(* CODESYS project pmps3.5.0.library
   Company: SLAC - LCLS
   DefaultNamespace: PMPS
   Version: 3.5.0
   Description: Collection of PMPS functionality for LCLS PLCs
   Placeholder: PMPS
   Author: Alex Wallace and contributors
   Title: PMPS

Project tree, tasks and I/O mapping:
  libraries: LCLS General, * (SLAC); Tc2_MC2, * (Beckhoff Automation GmbH); Tc2_Standard, * (Beckhoff Automation GmbH); Tc2_System, * (Beckhoff Automation GmbH); Tc2_Utilities, * (Beckhoff Automation GmbH); Tc3_JsonXml, * (Beckhoff Automation GmbH); Tc3_Module, * (Beckhoff Automation GmbH); TcUnit, 1.2.0.0 (www.tcunit.org)
  AncillaryComponents/
    function block FB_JsonDocToSafeBP [ST]: ACT_FFO, ACT_Logger, M_LoadSafeBP
    function block FB_JsonFileToJsonDoc [ST]: ACT_FFO, ACT_Logger
    function block FB_PressSensor_FFO [ST]: ACT_Logger
    function block FB_TempSensor_FFO [ST]: ACT_Logger
  DUTs/
    InternalDUT/
      data type E_MPSBeamClasses
      data type E_MPSBeamRates
      data type K_Apertures
      data type K_Attenuators
      data type K_Stopper
      data type L_Apertures
      data type L_Attenuators
      data type L_Stopper
      data type ST_AttenuatorStatus
      data type ST_BP_ArbInternal
      data type ST_FF
      data type ST_FFInfo
      data type ST_FFOverride
      data type ST_PMPS_Aperture
      data type ST_PMPS_Attenuator
      data type T_HashTableEntry
    UserDUT/
      data type ST_BeamParams
      data type ST_DbStateParams
      data type ST_Device
      data type ST_ReactiveParams
    data type PMPS_CODES
    data type ST_DeviceState
    data type ST_DeviceStateExt
    data type ST_DeviceStateTable
  GVLs/
    global variables PMPS_GVL
    global variables PMPS_PARAM
    global variables PMPS_TOOLS
  HelperFunctions/
    TypeTranslators/
      function APT_TO_IO [ST]
      function ATT_TO_IO [ST]
      function BP_TO_IO [ST]
      function F_DeviceState_To_DeviceStateExt [ST]
      function IO_TO_APT [ST]
      function IO_TO_ATT [ST]
      function IO_TO_BP [ST]
    function F_AttenuatorOK [ST]
    function F_BPWithID [ST]
    function F_DifferentBeamParams [ST]
    function F_eVExcludeRange [ST]
    function F_eVIncludeRange [ST]
    function F_eVRangeCalculator [ST]
    function F_eVWithinSpec [ST]
    function F_InitTestBP [ST]
    function F_PMPS_JSON [ST]
    function F_SafeBPCompare [ST]
    function F_SafeBPCompare0Rate [ST]
    function F_SetBeamParams [ST]
    function F_SetGoodAttStatus [ST]
    function F_SetStateParams [ST]
    function F_ValidReqID [ST]
    function block FB_DummyArbIO [ST]: ApplyBPReq, AutoUpdateBP, CheckRequest, RemoveRequest, RequestBP, ElevateRequest, nLowerAuthorityID
    function block FB_DummyHA [ST]: CheckRequest, ElevateRequest, nLowerAuthorityID, RemoveRequest, RequestBP
    function block PE_Ranges [ST]: FB_init
  ImplicitChecks/
    function CheckBounds [ST]
    function CheckDivDInt [ST]
    function CheckDivLInt [ST]
    function CheckDivLReal [ST]
    function CheckDivReal [ST]
    function CheckLRangeSigned [ST]
    function CheckLRangeUnsigned [ST]
    function CheckPointer [ST]
    function CheckRangeSigned [ST]
    function CheckRangeUnsigned [ST]
  MajorComponents/
    Arbiter/
      function block FB_Arbiter [ST]: AddRequest, ArbitrateBP, CheckRequest, CheckRequestInPool, ElevateRequest, FB_init, GetArbitratedBP, nEntryCount, nLowerAuthorityID, RemoveRequest, RequestBP
      function block FB_BeamParamAssertionPool [ST]: A_Add, A_Count, A_GetFirst, A_GetNext, A_Lookup, A_Remove, A_Reset, DataPoolToEpics
      function block FB_VetoArbiter [ST]: CheckRequest, RemoveRequest, RequestBP
    BPTM/
      function block BeamParameterTransitionManager [ST]: AssertFinalBP, AssertTransitionBP, AuthorizeTransition, DeauthorizeTransition, LogActions, NewTarget_ENTRY, RemoveTransitionAssertion, RequestBP_DO, SetNewTarget, WaitingForFinalAssertion_DO, WaitingForFinalAssertion_EXIT, WaitingForTransitionAssertion_DO, WaitingForTransitionAssertion_EXIT
      data type E_BPTMState
    FastFaults/
      function block FB_FastFault [ST]
      function block FB_HardwareFFOutput [ST]: EvaluateOutput, EvaluateOverrides, EvaluateVetos, Execute, ExecuteLogging, ExecuteNoLog, FormulateLogJson, IdxCheckIn, Register
    InterPlcComm/
      function block FB_ArbiterToSubSys_IO [ST]
      function block FB_SubSysToArbiter_IO [ST]: CheckRequest, RemoveRequest, RequestBP
    PhotonEnergyInterface/
      function F_CalculatePhotonEnergy [ST]
      function block FB_AcceleratorLinks [ST]
      function block FB_Hgvpu [ST]: Init, rCurrentPhotonEnergy, rTargetPhotonEnergy, UndAdrUpdate
      function block FB_KPhotonEnergy [ST]
      function block FB_LPhotonEnergy [ST]
      function block FB_PhotonEnergy [ST]
      function block FB_SXU [ST]: Init, rCurrentPhotonEnergy, rTargetPhotonEnergy, UndAdrUpdate
      function block FB_UndulatorSegment [ST]
    PMPS_MPS_Interface/
      function block FB_BeamClassOutputs [ST]
      function block FB_BeamClassOutputs_BCD [ST]
      function block FB_BeamClassWatcher [ST]
      function block FB_CTLS_Outputs [ST]
      function block FB_MachineModeFromEPICS [ST]
      function block FB_PhotonEnergyWatcher [ST]
    SimulationFB/
      function block FB_eVSimulator [ST]
      function block FB_MachineSimulator [ST]
    Stoppers/
      function block FB_KStopper [ST]: FB_init
      function block FB_KVetoDevice [ST]: FB_init
      function block FB_LStopper [ST]: FB_init
      function block FB_LVetoDevice [ST]: FB_init
      function block FB_StopperWatcher [ST]
      function block FB_VetoDevice [ST]
    function block FB_BeamClassFromEPICS [ST]
    function block FB_BPControlDevice [ST]: FB_init
    function block FB_BPRequestor [ST]: CheckRequest, RemoveRequest, RequestBP
    function block FB_LinearDeviceStateTable [ST]: A_Add, A_Count, A_GetFirst, A_GetNext, A_Lookup, A_Remove, A_Reset
    function block FB_LinearGovernor [ST]
    function block FB_RateFromEPICS [ST]
    interface I_HigherAuthority: CheckRequest, RemoveRequest, RequestBP
    interface I_LowerAuthority: ElevateRequest, nLowerAuthorityID
    interface I_UndulatorComplex: rCurrentPhotonEnergy, rTargetPhotonEnergy
  TestComponents/
    DUT/
      data type E_ArbDosTestStates
      data type E_BPTMTestStates
    function block FB_Arbiter_Test [ST]: ArbiterCapacity, Arbitration, DoS, FullArbitrationStack, RemoveReq, RequestCheckRemoveBP, StackArbiters
    function block FB_ArbToSubsys_Test [ST]: BasicFunction
    function block FB_AttenuatorSimulator [ST]
    function block FB_BPTM_Test [ST]: BPTMBasicFunction, FullArbError, InterruptAtAllSteps
    function block FB_DiffBP_Test [ST]: BPDiff
    function block FB_evRangeCalculator_Test [ST]: BasicFunction
    function block FB_eVWithinSpec_Test [ST]: evWithinRangeChecks
    function block FB_FastFault_Test [ST]: FFCombinedFunctionality, FFOvrdAndNextFault, FFRegistration
    function block FB_PhotonEnergyWatcher_Test [ST]: PEWatcherBasicFunction
    function block FB_SafeBPCompare_Test [ST]: BeamOffIsSafe, BPComparisonCheck
    function block FB_SubsysToArb_Test [ST]: BasicFunction, VetoFunction
    function block FB_VetoArbiter_Test [ST]: VetoArbiter
  VISUs/
  program MAIN [ST]
*)

// DUTs/InternalDUT/E_MPSBeamClasses

TYPE E_MPSBeamClasses :
(
    Beam_Off    :=  0,
    Kicker_STBY :=  1,
    BC1Hz       :=  2,
    BC10Hz      :=  3,
    Diagnostic  :=  4,
    BC120Hz     :=  5,
    Tuning      :=  6,
    MAP_1       :=  7,
    MAP_5       :=  8,
    MAP_10      :=  9,
    MAP_25      := 10,
    MAP_50      := 11,
    MAP_100     := 12,
    FULL        := 13,
    SPARE1      := 14,
    SPARE2      := 15
);
END_TYPE

// DUTs/InternalDUT/E_MPSBeamRates

TYPE E_MPSBeamRates :
(
    MPSRateInvalid            :=  0,
    MPSRate0Hz                :=  1,
    (* Previously used 2 and 3 for single shot and burst *)
    MPSRate1Hz                :=  4,
    MPSRate10Hz               :=  5,
    MPSRate30Hz               :=  6,
    MPSRate60Hz               :=  7,
    MPSRate120Hz              :=  8,
    MPSRateUnknown            :=  9,
    MPSRateSingleShot         := 10,
    MPSRateBurstMode          := 11,
    MPSRateBurstModeNotActive := 12,
    MPSNumberOfBeamRates      := 13,
    MPSRateBurstInvalid       := 14
)UINT;
END_TYPE

// DUTs/InternalDUT/K_Apertures
{attribute 'qualified_only'}
{attribute 'strict'}
{attribute 'to_string'}
TYPE K_Apertures :
(
    SL1K0 := 1,
    SL2K0 := 2
);
END_TYPE

// DUTs/InternalDUT/K_Attenuators
{attribute 'qualified_only'}
{attribute 'strict'}
TYPE K_Attenuators :
(
    AT1K0 := 1, // FEE Gas Attenuator
    AT1K4 := 2, // TMO Solid Attenuator in the FEE
    AT1K2 := 3, // RIX Solid Attenuator
    AT2K2 := 4, // RIX Solid Attenuator
    AT1K3 := 5 // TXI Solid Attenuator
);
END_TYPE

// DUTs/InternalDUT/K_Stopper
{attribute 'qualified_only'}
{attribute 'strict'}
TYPE K_Stopper :
(
    ST3K4 := 1, // TMO PPS stopper in
    ST1K2 := 2, // RIX PPS stopper in
    MR1K1_IN := 3, // Monochromator focus optic vertical state
    MR1K1_OUT := 4, // Monochromator focus optic vertical state
    MR1K3_IN := 5, // TXI MR1K3 Offset Mirror horizontal state
    MR1K3_OUT := 6, // TXI MR1K3 Offset Mirror horizontal state
    ST4K4 := 7, //TMO ST4K4 Photon Terminator In Limit Switch
    ST1K4 := 8, //TMO Photon Stopper in the FEE
    ST1K3 :=9, //TXI Kline PPS stopper in
    MR2K3_IN := 10, // TXI MR2K3 Offset Mirror state
    MR2K3_OUT := 11, // TXI MR2K3 Offset Mirror horizontal state
    DEFAULT := PMPS_GVL.MAX_VETO_DEVICES // DO NOT USE FOR ANYTHING
);
END_TYPE

// DUTs/InternalDUT/L_Apertures
{attribute 'qualified_only'}
{attribute 'strict'}
{attribute 'to_string'}
TYPE L_Apertures :
(
    SL1L0 := 1,
    SL2L0 := 2
);
END_TYPE

// DUTs/InternalDUT/L_Attenuators
{attribute 'qualified_only'}
{attribute 'strict'}
{attribute 'to_string'}
TYPE L_Attenuators :
(
    AT1L0 := 1, // FEE Combo Gas/Solid Attenuator
    AT2L0 := 2 // FEE Solid Attenuator
);
END_TYPE

// DUTs/InternalDUT/L_Stopper
{attribute 'qualified_only'}
{attribute 'strict'}
TYPE L_Stopper :
(
    ST1L0 := 1, // ST1
    ST1L1 := 2, // TXI PPS Stopper in
    MR1L0_L0 := 3, // MR1L0 Pitch state delivery to L0 line
    MR1L0_TXI := 4, //MR1L0 Pitch state delivery to TXI line
    MR1L1_IN:= 5, //  TXI Offset Mirror horizontal state
    MR1L1_OUT:= 6, // TXI Offset Mirror horizontal state
    DEFAULT := PMPS_GVL.MAX_VETO_DEVICES // DO NOT USE FOR ANYTHING
);
END_TYPE

// DUTs/InternalDUT/ST_AttenuatorStatus
TYPE ST_AttenuatorStatus :
STRUCT
    AtTarget : BIT;     //0
    Moving : BIT;       //1
    LocalMode : BIT;    //2  (* means the attenuator ignores PMPS preemptive requests and operates from a local setpoint *)
    PMPSMode : BIT;     //3  (* means the attenuator is only taking setpoints from the pmps *)
    OK : BIT;           //4
    Toggle : BIT;       //5  just here for fun
    Include : BIT;      //6  Consider this device status
END_STRUCT
END_TYPE

// DUTs/InternalDUT/ST_BP_ArbInternal
TYPE ST_BP_ArbInternal EXTENDS ST_BeamParams :
STRUCT
    {attribute 'pytmc' := 'pv: ID
        io: i
    '}
    nId : DWORD;
    {attribute 'pytmc' := 'pv: Live
        io: i
    '}
    LiveInTable : BOOL;
    {attribute 'pytmc' := 'pv: Device
        io: i
    '}
    sDevName: STRING;
END_STRUCT
END_TYPE

// DUTs/InternalDUT/ST_FF
TYPE ST_FF :
STRUCT
    {attribute 'pytmc' := '
        pv: Info
     '}
    Info : ST_FFInfo;

    {attribute 'pytmc' := '
        pv: Ovrd
     '}
    Ovrd : ST_FFOverride;

    {attribute 'pytmc' := '
        pv: OK
        io: i
     '}
    OK   :   BOOL; // Fault logic state

    FaultAck : BOOL; // Set when faulted, reset by logger.
    ClearAck : BOOL;

    {attribute 'pytmc' := '
        pv: BeamPermitted
        io: i
     '}
    BeamPermitted   :   BOOL; // Result of reset, veto, and fault logic, true beam off boolean

    {attribute 'pytmc' := '
        pv: Reset
        io: o
     '}
    Reset   :   BOOL;

    bsFF    :    RS;
    rtReset    :    R_TRIG;
    ftCountFault : F_TRIG;

END_STRUCT
END_TYPE

// DUTs/InternalDUT/ST_FFInfo

// These elements should be set at init and never changed.

TYPE ST_FFInfo :
STRUCT
    {attribute 'pytmc' := '
        pv: Path
        io: i
     '}
    sPath   :    T_MaxString; // Full PLC path to FF object
    {attribute 'pytmc' := '
        pv: Desc
        io: i
     '}
    Desc    :   T_MaxString; // Set at instantiation to a helpful description of the fast fault purpose
    {attribute 'pytmc' := '
        pv: DevName
        io: i
     '}
    DevName :   T_MaxString; // Component name, used in diagnostic to help narrow down where beam faults are coming from
    {attribute 'pytmc' := '
        pv: TypeCode
        io: i
     '}
    TypeCode    :   UINT; // Set at instantiation to fault class code

///////////////////////////////////////////
// Warning, this variable is effectively a VETO of the fast fault if set FALSE
// Do not alter the state of this variable unless you really know what you're doing.
///////////////////////////////////////////
    {attribute 'pytmc' := '
        pv: InUse
        io: i
     '}
    InUse   :   BOOL := FALSE; // If this FF is currently in-use
///////////////////////////////////////////


    AutoReset   :   BOOL; // Automatically clear fast fault (latching vs non-latching)
    Vetoable  : BOOL := TRUE; // Can this fast fault be masked by the veto device input?

      {attribute 'pytmc' := '
        pv: InfoString
        io: i
     '}
    InfoString : STRING;
END_STRUCT
END_TYPE

// DUTs/InternalDUT/ST_FFOverride
TYPE ST_FFOverride :
STRUCT
    {attribute 'pytmc' := '
        pv: Duration
        io: o
     '}
    Duration : DINT; // DINT to be compatible with EPICS

    {attribute 'pytmc' := '
        pv: Expiration
        io: o
     '}
    Expiration : DINT; // DINT to be compatible with EPICS

    {attribute 'pytmc' := '
        pv: StartDT
        io: o
     '}
    StartDT : DINT; // DINT to be compatible with EPICS

    {attribute 'pytmc' := '
        pv: Activate
        io: o
     '}
    Activate : BOOL;

    {attribute 'pytmc' := '
        pv: Deactivate
        io: o
     '}
    Deactivate : BOOL;

    {attribute 'pytmc' := '
        pv: ElapsedTime
        io: i
     '}
    ElapsedTime : DINT; // DINT to be compatible with EPICS

    {attribute 'pytmc' := '
        pv: RemainingTime
        io: i
     '}
    RemainingTime : DINT; // DINT to be compatible with EPICS

    {attribute 'pytmc' := '
        pv: Active
        io: i
     '}
    Active: BOOL;

    Timer    :   TP;
    OvrdActLogAck : BOOL;
    OvrdExpLogAck : BOOL;

    tOvrdActivate : R_TRIG;
    tOvrdExpiring  : F_TRIG;
END_STRUCT
END_TYPE

// DUTs/InternalDUT/ST_PMPS_Aperture
TYPE ST_PMPS_Aperture EXTENDS ST_PMPS_Aperture_IO :
STRUCT
    (*
    {attribute 'pytmc' := 'pv: Width
            io: i
            field: EGU mm'}
    Width : REAL; // distance between horizontal slits (x)
    {attribute 'pytmc' := 'pv: Height
            io: i
            field: EGU mm'}
    Height : REAL; // distance between vertical slits (y)

    {attribute 'pytmc' := 'pv: OK
        io: i'}
    xOK : BOOL; // status of aperture, false if error or in motion
    *)
END_STRUCT
END_TYPE

// DUTs/InternalDUT/ST_PMPS_Attenuator
TYPE ST_PMPS_Attenuator EXTENDS ST_PMPS_Attenuator_IO :
STRUCT
    (*
        {attribute 'pytmc' := 'pv: Att
            io: i
            field: EGU %
        '}
        nTran : UINT;
        {attribute 'pytmc' := 'pv: OK
            io: i
        '}
        xAttOK : UINT; // true = no errors and attenuator is stable
        *)
END_STRUCT
END_TYPE

// DUTs/InternalDUT/T_HashTableEntry
TYPE T_HashTableEntry :
STRUCT
    {attribute 'pytmc' := '
        pv: Key
        io: i
     '}
    key : DWORD := 0;
    value : PVOID := 0;
END_STRUCT
END_TYPE

// DUTs/UserDUT/ST_BeamParams
TYPE ST_BeamParams :
    STRUCT
        (*  Requested pre-optic attenuation %  *)
        {attribute 'pytmc' := 'pv: Transmission
            io: i
            field: HOPR 1;
            field: LOPR 0;
            field: PREC 2;
        '}
        nTran : REAL := 0;
        (* Pulse-rate *)
        {attribute 'pytmc' := 'pv: Rate
            io: i
            field: EGU Hz
        '}
        nRate : UDINT := 0;
        (* Photon energy ranges *)
        {attribute 'pytmc' := 'pv: eVRanges
            io: i
            field: EGU eV'}
        {attribute 'displaymode' := 'binary'}
        neVRange : DWORD := 0;
                 (* Photon energy  *)
        {attribute 'pytmc' := 'pv: PhotonEnergy
            io: i
            field: EGU eV'}
        neV : REAL := 0;
        (* Beamclass ranges *)
         {attribute 'pytmc' := 'pv: BeamClassRanges
            io: i'}
        {attribute 'displaymode' := 'binary'}
        nBCRange : WORD := 0;
        (* Beamclass *)
        {attribute 'pytmc' := 'pv: BeamClass
            io: i'}
        nBeamClass : USINT :=0;
        (* Machine Mode *)
        {attribute 'pytmc' := 'pv: MachineMode
            io: i'}
        nMachineMode: USINT:=3;
        (* Beamline attenuators *)
        {attribute 'pytmc' := 'pv: AuxAtt
        io: i'}
        astAttenuators : ARRAY [1..PMPS_GVL.AUX_ATTENUATORS] OF ST_PMPS_Attenuator;

        (* Stoppers *)
        {attribute 'pytmc' := 'pv: Veto
        io: i'}
        aVetoDevices : ARRAY [1..PMPS_GVL.MAX_VETO_DEVICES] OF BOOL;

        (* Apertures *)
        {attribute 'pytmc' := 'pv: Apt
        io: i'}
        astApertures : ARRAY [1..PMPS_GVL.MAX_APERTURES] OF ST_PMPS_Aperture := [(Width:=1E3, Height:=1E3), (Width:=1E3, Height:=1E3),(Width:=1E3, Height:=1E3),(Width:=1E3, Height:=1E3)];

        // Toggle for watchdog
        xValidToggle : BOOL;
        // Beam parameter set is valid (if readback), or acknowledged (if request)
        {attribute 'pytmc' := 'pv: Valid
        io: i'}
        xValid : BOOL;
        // Cohort index. Identifies which cohort this BP set was included in arbitration
        {attribute 'pytmc' := 'pv: Cohort
        io: i
            field: DESC Cohort inc on each arb cycle
        '}
        nCohortInt : UDINT;
    END_STRUCT
END_TYPE

// DUTs/UserDUT/ST_DbStateParams
TYPE ST_DbStateParams :
     // Defines The parameters that are loaded from the json db for every state name
STRUCT
      // PMPS database lookup name for this state
    {attribute 'pytmc' := '
        pv: PMPS_STATE
        io: i
        field: DESC PMPS Database Lookup Key
    '}
    sPmpsState: STRING;

    // Beam parameters associated with this state
    {attribute 'pytmc' := '
        pv: BP
        io: i
    '}
    stBeamParams: ST_BeamParams := PMPS_GVL.cst0RateBeam;

    // Set to TRUE once the PMPS library has loaded a valid state from the database
    {attribute 'pytmc' := '
        pv: PMPS_LOADED
        io: i
        field: DESC TRUE if PMPS loaded parameters from the database.
    '}
    bBeamParamsLoaded: BOOL;

     // Reactive parameters associated with this state
    {attribute 'pytmc' := '
        pv: ReParams
        io: i
    '}
    stReactiveParams : ST_ReactiveParams;

    // Transition ID associated with this state
    {attribute 'pytmc' := '
        pv: PMPS_ID
        io: i
        field: DESC Assertion Request ID
    '}
    nRequestAssertionID: UDINT;
END_STRUCT
END_TYPE

// DUTs/UserDUT/ST_Device
TYPE ST_Device :
STRUCT
    //IO
    stAxis	:	AXIS_REF;
    //The following limit switches must be TRUE or high (ie. NC) to enable that direction of motion
    //The EPICS display should show an inverted indicator to communicate end of travel reached
    i_xLoLim	AT %I*	:	BOOL; //Wire normally-closed
    i_xHiLim	AT %I*	:	BOOL; //Wire normally-closed

    //Acuator Parameters
    lrUpperPositionLimit	:	LREAL := 10000000000; //Use in conjuntion with limit switches or set to a huge number to ignore
    lrLowerPositionLimit	:	LREAL := -10000000000; //Use in conjuntion with limit switches or set to a huge number to ignore

    xEnable	:	BOOL := TRUE;

    //Supervisory System

    //MPS Override
    xOverrideMPSLimits	: BOOL := FALSE; //Set true to move beyond MPS limits. Note this will trip beam off.

    //Status and Faults
    xClearFaults	:	BOOL;	//Rising edge tries to clear faults of all kinds

    xGovernorFault	:	BOOL;	//Indicates governor is faulted
    xGovernorOverridden	:	BOOL; //Indicates governor is in override mode
    xSMFault		:	BOOL;	//Indicates component state machine is faulted

    //Device States
    StateTable		:	FB_LinearDeviceStateTable;

    stTransitionState	:	ST_DeviceState; //The transition state might have non-zero beam parameters
    nSafeState			:	UDINT; //State where the device is considered safe
    nTransitionState	:	UDINT;

    nRequestedState	:	UDINT; //EPICS control, cleaned (checked against array limits) and deposited in nTargetState
    nTargetState	:	UDINT; //The requested state should be deposited here after cleaning
    nActiveState	:	UDINT; //The last successfully reached state


END_STRUCT
END_TYPE

// DUTs/UserDUT/ST_ReactiveParams
TYPE ST_ReactiveParams :
STRUCT
    {attribute 'pytmc' := 'pv: TempSP
            io: i
            field: PREC 2;
            field: EGU "C";
        '}
    nTempSP: REAL;
    {attribute 'pytmc' := 'pv: PressSP
            io: i
            field: PREC 2;
            field: EGU "TORR";
        '}
    nPressSP: REAL;
END_STRUCT
END_TYPE

// DUTs/PMPS_CODES
{attribute 'qualified_only'}
{attribute 'strict'}
TYPE PMPS_CODES :
(
    FAST_FAULT := 16#1, // Generic fast fault
    PEW_FAULT := 16#7, // Fault occurs when the calculated machine photon energy (K value calculated by undulator gap, and electron energy) falls outside the permitted range.

    // Arbiter codes
    //////////////////////////////////
        ARB_FULL := 16#201, // Arbiter pool is full.

    //BPTM Codes
    //////////////////////////////////
        BadTargetID := 16#300,
        BadTransID := 16#301,
        TransAssrtFail := 16#302,
        FinalAssrtFail := 16#303,
        NoRoomInArb := 16#304
) UINT;
END_TYPE

// DUTs/ST_DeviceState
TYPE ST_DeviceState :
STRUCT

    //State name
    sStateName	:	STRING;
    nStateRef	:	UDINT; //Primary key of device state database

    //////////////////
    // This stuff may belong in a sub-class or something
    //Position
    rPosition	:	REAL := 0; //Center of the state
    //Tolerance
    rTolerance :	REAL := 0; //+/- amount
    //////////////////
    //Required beam parameters
    stReqBeamParam	:	ST_BeamParams;

END_STRUCT
END_TYPE

// DUTs/ST_DeviceStateExt
//Use when working with states in code
//Extended with a valid boolean to indicate the structure was loaded
//properly
TYPE ST_DeviceStateExt EXTENDS ST_DeviceState :
STRUCT
    xValid	:	BOOL := FALSE;
END_STRUCT
END_TYPE

// DUTs/ST_DeviceStateTable
TYPE ST_DeviceStateTable :
STRUCT
    iDeviceID:DINT;
    iStateID:DINT;
    rTargetPosition: REAL;
    rTolerance: REAL;
    rTransmission: REAL;
    iBeamClass : DINT;
    iPulseRate: DINT;
    rPerPulseEnergy:REAL;
    rUpper_eV: REAL;
    rLower_eV: REAL;
    rPhotonEnergy: REAL;
END_STRUCT
END_TYPE

// MajorComponents/BPTM/E_BPTMState
TYPE E_BPTMState :
(
    Init := 0,
    NewTarget := 1000,
    RequestBP := 1500,
    WaitForBP := 2500,
    WaitingForTransitionAssertion := 2000,
    WaitingForFinalAssertion := 3000,
    Transitioning := 4000,
    WaitForFinalBP := 5000,
    CleaningUp := 6000,
    Idle := 10000,
    Done := 8000,
    Error := 9000
);
END_TYPE

// TestComponents/DUT/E_ArbDosTestStates
{attribute 'qualified_only'}
{attribute 'strict'}
TYPE E_ArbDosTestStates :
(
    Init := 0,
    SecondReq := 100,
    WaitForAck := 200,
    WaitFor2ndAck := 300,
    RunAsserts := 8000
);
END_TYPE

// TestComponents/DUT/E_BPTMTestStates
{attribute 'qualified_only'}
{attribute 'strict'}
TYPE E_BPTMTestStates :
(
    Init := 0,
    WaitingForValidID := 50,
    WaitingForTransitionAssertion := 100,
    StalledAtTransition := 150,
    WaitingForFinalAssertion    := 200,
    WaitingForBeam := 250,
    Transitioning    := 300,
    CleaningUp    := 400,
    AnotherState := 500,
    Retry := 1000,
    Done := 8000,
    Error := 9000
);
END_TYPE

// GVLs/PMPS_GVL
{attribute 'qualified_only'}
VAR_GLOBAL
    {attribute 'pytmc' := '
        pv: @(PREFIX)RequestedBP
        io: i
        archive: 1Hz monitor
    '}
    stRequestedBeamParameters    :    ST_BeamParams; //Summarized request for the line, as recognized by the line arbiter PLC
    {attribute 'pytmc' := '
        pv: @(PREFIX)CurrentBP
        io: i
        archive: 1Hz monitor
    '}
    stCurrentBeamParameters    :    ST_BeamParams; //Currently active BP set, broadcast by the line arbiter PLC

    {attribute 'pytmc' := '
        pv: @(PREFIX)eVRangeCnst
        io: i
        archive: 1Hz monitor
        field: DESC Active eV Range constants
        field: EGU eV
    '}
    g_areVBoundaries    :    ARRAY [0..g_cBoundaries]    OF    REAL;



    PERange : PE_Ranges; //Included to place the ev ranges properly
END_VAR
VAR_GLOBAL RETAIN
    // Statistics
    {attribute 'pytmc' := '
        pv: @(PREFIX)SuccessfulPreemptions
        io: i
    '}
    SuccessfulPreemption : UDINT; // Any time BPTM applies a new BP request which is confirmed
    {attribute 'pytmc' := '
        pv: @(PREFIX)AccumulatedFastFaults
        io: i
    '}
    AccumulatedFF : UDINT; // Any time a FF occurs
    BP_jsonDoc 		: SJsonValue;
END_VAR
VAR_GLOBAL CONSTANT

    EXCLUDED_ASSERTION_ID    :    UDINT    := 16#FFFFFFFF; //An assertion ID that should always return "not found" in the assertion pool
    VISIBLE_TEST_VELOCITY    :    LREAL    := 10;
    FAST_TEST_VELOCITY        :    LREAL    := 100;
    MAX_DEVICE_STATES        :    UDINT    := 300;

    TRANS_SCALING_FACTOR : REAL := REAL#1.0; // Scaling factor for fixed-point transmission

    AUX_ATTENUATORS : UINT := 16; // Maximum # of attenuators in the PMPS
    MAX_VETO_DEVICES   :   UINT := 16;
    stAttenuators : ST_PMPS_Attenuator :=(nTran:=1,xAttOK:=1);
    {attribute 'pytmc' := '
        pv: @(PREFIX)FullBeamCnst
        io: i
        archive: 1Hz monitor
        field: DESC Full beam constant
    '}
    cstFullBeam    :    ST_BeamParams := (
        nTran := 1,
        neVRange :=  2#1111_1111_1111_1111_1111_1111_1111_1111,
        nRate    := UDINT#1000000,
        nBCRange := 2#0111_1111_1111_1111,
        astApertures := [(Width:=1E3, Height:=1E3), (Width:=1E3, Height:=1E3),(Width:=1E3, Height:=1E3),(Width:=1E3, Height:=1E3)],
        astAttenuators :=  [PMPS_GVL.AUX_ATTENUATORS(stAttenuators)]

    );
    {attribute 'pytmc' := '
        pv: @(PREFIX)0RateBeamCnst
        io: i
        archive: 1Hz monitor
        field: DESC 0-rate beam constant
    '}
    cst0RateBeam    :    ST_BeamParams := ( // Use for transition requests
        nTran := 1,
        neVRange :=  2#1111_1111_1111_1111_1111_1111_1111_1111,
        nRate    := 0,
        nBCRange := 2#0000_0000_0000_0000,
        astApertures := [(Width:=1E3, Height:=1E3), (Width:=1E3, Height:=1E3),(Width:=1E3, Height:=1E3),(Width:=1E3, Height:=1E3)],
        astAttenuators :=  [PMPS_GVL.AUX_ATTENUATORS(stAttenuators)]
    );
   (*  {attribute 'pytmc' := '
        pv: @(PREFIX)SafeBeamCnst
        io: i
        archive: 1Hz monitor
        field: DESC Safe beam constant
    '}
   cstSafeBeam    :    ST_BeamParams := (
        nTran := 0,
        neVRange := 0,
        nRate    := 0
    );*)

    cnMaxStateArrayLen : INT := 20;


    MAX_APERTURES : UINT := 4; // Maximum # of power slits in the PMPS
    {warning disable C0228}
    DUMMY_AUX_ATT_ARRAY : ARRAY [1..PMPS_GVL.AUX_ATTENUATORS] OF ST_PMPS_Attenuator;
    {warning restore C0228}



    g_cBoundaries    :    INT    := 31;


//////////////////////////
// L Undulator constants
//////////////////////////

///////////////////////////////////////

    {attribute 'pytmc' := '
        pv: @(PREFIX)eVRangeHyst
        io: i
        archive: 1Hz monitor
        field: DESC eV Range hystersis
        field: EGU eV
    '}
    reVHyst: REAL := 5; //


    {attribute 'pytmc' := '
        pv: @(PREFIX)L:eVRangeCnst
        io: i
        archive: 1Hz monitor
        field: DESC eV Range constants
        field: EGU eV
    '}
    g_areVBoundariesL    :    ARRAY [0..g_cBoundaries]    OF    REAL    := [
    1.0E3,
    1.7E3,
    2.1E3,
    2.5E3,
    3.8E3,
    4.0E3,
    5.0E3,
    7.0E3,
    7.5E3,
    7.7E3,
    8.9E3,
    10.0E3,
    11.1E3,
    12.0E3,
    13.0E3,
    13.5E3,
    14.0E3,
    16.9E3,
    18.0E3,
    20.0E3,
    22.0E3,
    24.0E3,
    25.0E3,
    25.5E3,
    26.0E3,
    27.0E3,
    28.0E3,
    28.5E3,
    29.0E3,
    30.0E3,
    60.0E3,
    90.0E3
    ];


    {attribute 'pytmc' := '
        pv: @(PREFIX)K:eVRangeCnst
        io: i
        archive: 1Hz monitor
        field: DESC eV Range constants
        field: EGU eV
    '}
    g_areVBoundariesK    :    ARRAY [0..g_cBoundaries]    OF    REAL    := [
    100,
    250,
    270,
    350,
    400,
    450,
    480,
    530,
    680,
    730,
    850,
    1.10E3,
    1.15E3,
    1.25E3,
    1.45E3,
    1.50E3,
    1.55E3,
    1.65E3,
    1.70E3,
    1.75E3,
    1.82E3,
    1.85E3,
    2.00E3,
    2.20E3,
    2.50E3,
    2.80E3,
    3.00E3,
    3.15E3,
    3.50E3,
    4.00E3,
    5.30E3,
    7.00E3
    ];


END_VAR

// GVLs/PMPS_PARAM
{attribute 'qualified_only'}
VAR_GLOBAL CONSTANT
    MAX_FAST_FAULTS	:	UINT := 50; // Max fast faults for an FFO
    MAX_ASSERTIONS    :    UDINT := 20; //Maximum number of BP requests in the arbiter
    TRANS_MARGIN : REAL := REAL#0.05; // Allowed % margin above requested transmission level in SafeBPCompare (0.0500 = 5deci% default). Note: change this value if scaling factor changes.
END_VAR

// GVLs/PMPS_TOOLS
{attribute 'qualified_only'}
VAR_GLOBAL
    fbJson : FB_JsonSaxWriter;
END_VAR

// AncillaryComponents/FB_JsonDocToSafeBP
FUNCTION_BLOCK FB_JsonDocToSafeBP
VAR_INPUT
    bExecute             : BOOL; //Rising Edge
    jsonDoc 		: SJsonValue;
    sDeviceName : STRING;
END_VAR
VAR_OUTPUT
    bHasDevice		: BOOL;
    bHasAllStates		: BOOL;
    bHasAllParameters :BOOL := TRUE;
    bBusy                : BOOL;
    bError               : BOOL;
    nErrId               : UDINT;
    sErrMsg				 :STRING;
END_VAR
VAR_IN_OUT
    //ARRAY [1.. MOTION_GVL.MAX_STATES] ;
    arrStates: ARRAY[*] OF ST_DbStateParams;
    io_fbFFHWO    :    FB_HardwareFFOutput;
END_VAR
VAR
    (* JSON *)
    fbJson 			: FB_JsonDomParser;
    jsonProp		: SJsonValue;
    jsonValue		: SJsonValue;
    jsonParam		: SJsonValue;
    jsonnTran      : SJsonValue;
    jsonnRate      : SJsonValue;
    Step: INT;
    index: DINT;
    nStateCount:DINT;
    RisingEdge           : R_TRIG;

    (*Logger*)
    tNewMessage : R_TRIG;
    fbLogger : FB_LogMessage := (eSubsystem:=E_SubSystem.MPS, nMinTimeViolationAcceptable:=10);
    (*FFO*)
    FFO    :    FB_FastFault :=(
        i_Desc := 'Fault occurs when there is an error loading safe beam parameters from json file',
        i_TypeCode := 16#FF13);
    sbuffReadSmall: INT;
END_VAR

(* Retrieve JSON content *)
RisingEdge(CLK:=bExecute);

CASE Step OF
    0:     (* Idle state *)
          IF RisingEdge.Q THEN
               bBusy := TRUE;
               bError:= FALSE;
               nErrId:=0;
               sErrMsg :='';
               Step := 20;
               fbLogger(sMsg:='Start Parsing Json DOC.', eSevr:=TcEventSeverity.Info);
          END_IF

     20: (*Find the Device Name*)
        bHasDevice := fbJson.HasMember(jsonDoc, sDeviceName);
        IF (bHasDevice) THEN
            jsonProp := fbJson.FindMember(jsonDoc, sDeviceName);
            IF jsonProp <> 0 THEN
                Step := Step+1;
                ELSE
                    Step := 900 + Step;
                    nErrId := Step;
                    bError := TRUE;
                    sErrMsg:=  CONCAT('Error device name not found in Json File : ',sDeviceName);
                END_IF
        ELSE
            Step := 900 + Step;
            nErrId := Step;
            bError := TRUE;
            sErrMsg:=  CONCAT('Error device name not found in Json File : ',sDeviceName);
        END_IF

     21: (*Check device States in DOM*)
             nStateCount :=0;
             FOR Index:=LOWER_BOUND(arrStates,1) TO UPPER_BOUND(arrStates,1) BY 1 DO
                  IF NOT ((arrStates[Index].sPmpsState= '') OR (arrStates[Index].sPmpsState= 'Invalid')) THEN
                      IF NOT (fbJson.HasMember(jsonProp, arrStates[Index].sPmpsState)) THEN
                              Step := 900+ Step;
                              nErrId := Step;
                              bError := TRUE;
                              sErrMsg:= CONCAT('Error loading device state in Json File : ',arrStates[Index].sPmpsState);
                              fbLogger(sMsg:= sErrMsg, eSevr:=TcEventSeverity.Critical);
                              EXIT;
                        ELSE
                            nStateCount :=nStateCount+1;
                      END_IF
                   ELSE
                       bHasAllStates :=TRUE;
                       EXIT;
                  END_IF
            END_FOR

           Step := Step+1;

     22: //Make sure state array input has State name data
          IF (nStateCount =0) THEN
              bHasAllStates :=FALSE;
              Step := 900+ Step;
              nErrId := Step;
              bError := TRUE;
              sErrMsg:= CONCAT('Error Input State array is empty : ',sDeviceName);
         ELSE
             Step := Step+1;
         END_IF;

     23:  (*loop Device State Arrays to find load all States BP*)
          FOR Index:=LOWER_BOUND(arrStates,1) TO UPPER_BOUND(arrStates,1) BY 1 DO
              IF NOT (arrStates[Index].sPmpsState= '') THEN
                  IF(NOT M_LoadSafeBP(arrStates[Index].sPmpsState, Index)) THEN
                      Step := 900+ Step;
                      fbLogger.sMsg := CONCAT('Error Parsing beam parameters - Device/States: ', arrStates[Index].sPmpsState);
                      fbLogger(sMsg:= sErrMsg, eSevr:=TcEventSeverity.Critical);
                  END_IF
               ELSE
                    EXIT;
               END_IF
          END_FOR
          IF (bHasAllParameters) THEN Step := 30;
              ELSE Step := 900+ Step;
          END_IF

     30: (*ALL good here*)
         fbLogger.sMsg := CONCAT('Complete Parsing Json Doc. Device: ', sDeviceName);
        fbLogger.sMsg := CONCAT(fbLogger.sMsg ,' - States Count: ');
        fbLogger.sMsg := CONCAT(fbLogger.sMsg ,TO_STRING(nStateCount));
          fbLogger(eSevr:=TcEventSeverity.Info);
         bExecute:= FALSE;
        bBusy:=FALSE;
        Step := 0;
        FFO.i_xOK := TRUE;
END_CASE


//Fault in error state
IF(Step>=900) THEN
    FFO.i_xOK := FALSE;
    bBusy:=FALSE;
    Step:=0;
END_IF
ACT_FFO();
ACT_LOGGER();

ACTION ACT_FFO:
(*FAST FAULT*)
FFO(i_xOK := ,
    i_xReset := ,
    i_xAutoReset :=TRUE,
    i_DevName := sDeviceName,
    io_fbFFHWO := io_fbFFHWO);
END_ACTION

ACTION ACT_Logger:
// Log valve open
tNewMessage(CLK:= NOT(FbLogger.sMsg = sErrMsg) AND NOT (sErrMsg =''));
IF tNewMessage.Q THEN fbLogger(sMsg:= sErrMsg, eSevr:=TcEventSeverity.Critical); END_IF
END_ACTION

METHOD M_LoadSafeBP : BOOL
VAR_INPUT
    sStateName : STRING;
    Index:DINT;
END_VAR
VAR
    //bHasAllParameters : BOOL := TRUE;
    sAperture:STRING;
    nAperture:INT := -1;
    sEV:STRING;
    sBC:STRING;
    nIndex:INT;
END_VAR
bHasAllParameters :=  fbJson.HasMember(jsonProp, sStateName);
jsonValue := fbJson.FindMember(jsonProp, sStateName);
IF bHasAllParameters THEN
    //nTran
    bHasAllParameters R= NOT fbJson.HasMember(jsonValue, 'nTran');
    IF (NOT bHasAllParameters) THEN fbLogger(sMsg:= 'Error Loading nTran', eSevr:=TcEventSeverity.Critical); END_IF
    jsonnTran := fbJson.FindMember(jsonValue, 'nTran');
    arrStates[Index].stBeamParams.nTran := TO_REAL(fbJson.GetString(jsonnTran));

    //nRate
    bHasAllParameters R= NOT fbJson.HasMember(jsonValue, 'nRate');
    IF (NOT bHasAllParameters) THEN fbLogger(sMsg:= 'Error Loading nRate', eSevr:=TcEventSeverity.Critical); END_IF
    jsonnRate := fbJson.FindMember(jsonValue, 'nRate');
    arrStates[Index].stBeamParams.nRate:= TO_UDINT(fbJson.GetString(jsonnRate));

    //neVRange
    bHasAllParameters R= NOT fbJson.HasMember(jsonValue, 'neVRange');
    jsonParam := fbJson.FindMember(jsonValue, 'neVRange');
    sEV:=(fbJson.GetString(jsonParam));
    bHasAllParameters R= NOT (LEN(sEV)=32);
    This^.arrStates[Index].stBeamParams.neVRange :=0;
    IF (NOT bHasAllParameters) THEN
        fbLogger(sMsg:= 'Error Loading eVRange', eSevr:=TcEventSeverity.Critical);
        ELSE
            FOR nIndex := 0 TO PMPS_GVL.g_cBoundaries BY 1 DO
                This^.arrStates[Index].stBeamParams.neVRange := SHL(This^.arrStates[Index].stBeamParams.neVRange,1);
                This^.arrStates[Index].stBeamParams.neVRange := This^.arrStates[Index].stBeamParams.neVRange+HEXASCNIBBLE_TO_BYTE(sEV[nIndex]);
            END_FOR
    END_IF

    //nBeamClassRange
    bHasAllParameters R= NOT fbJson.HasMember(jsonValue, 'nBeamClassRange');
    jsonParam := fbJson.FindMember(jsonValue, 'nBeamClassRange');
    sBC:=(fbJson.GetString(jsonParam));
    bHasAllParameters R= NOT (LEN(sBC)=15);
    arrStates[Index].stBeamParams.nBCRange :=0;
    IF (NOT bHasAllParameters) THEN
            fbLogger(sMsg:= 'Error Loading Beam Class Range. Make sure Bitmask is equal than 15 bits.', eSevr:=TcEventSeverity.Critical);
    ELSE
        FOR nIndex := 0 TO 14 BY 1 DO
            arrStates[Index].stBeamParams.nBCRange := SHL(arrStates[Index].stBeamParams.nBCRange,1);
            arrStates[Index].stBeamParams.nBCRange := arrStates[Index].stBeamParams.nBCRange+HEXASCNIBBLE_TO_BYTE(sBC[nIndex]);
        END_FOR
     END_IF

    //ApertureName and Values
    bHasAllParameters R= NOT fbJson.HasMember(jsonValue, 'ap_name');
    jsonParam := fbJson.FindMember(jsonValue, 'ap_name');
    sAperture := fbJson.GetString(jsonParam);
{IF defined (L)}
    IF ('SL1L0' = sAperture) THEN nAperture := L_Apertures.SL1L0;
    ELSIF ('SL2L0' = sAperture) THEN nAperture := L_Apertures.SL2L0;
    END_IF
{ELSIF defined (K)} // Attribute 'to_string' only build 4024 TO_STRING(PMPS.K_Apertures.SL1K0) - need another non hardcoded way
    IF ('SL1K0' = sAperture) THEN nAperture := K_Apertures.SL1K0;
    ELSIF ('SL2K0' = sAperture) THEN nAperture := K_Apertures.SL2K0;
    END_IF
{END_IF}
    IF (nAperture>-1) THEN
        //Gap Height
        bHasAllParameters R= NOT fbJson.HasMember(jsonValue, 'ap_ygap');
        jsonParam := fbJson.FindMember(jsonValue, 'ap_ygap');
        arrStates[Index].stBeamParams.astApertures[nAperture].Height := TO_REAL(fbJson.GetString(jsonParam));

        //Gap Width
        bHasAllParameters R= NOT fbJson.HasMember(jsonValue, 'ap_xgap');
        jsonParam := fbJson.FindMember(jsonValue, 'ap_xgap');
        arrStates[Index].stBeamParams.astApertures[nAperture].Width := TO_REAL(fbJson.GetString(jsonParam));

        IF (NOT bHasAllParameters) THEN fbLogger(sMsg:= 'Error Loading aperture gap', eSevr:=TcEventSeverity.Critical); END_IF
    END_IF

    //Read Transition ID for the State
    bHasAllParameters R= NOT fbJson.HasMember(jsonValue, 'id');
    jsonParam := fbJson.FindMember(jsonValue, 'id');
    IF (NOT bHasAllParameters) THEN fbLogger(sMsg:= 'Error Loading Assertion ID', eSevr:=TcEventSeverity.Critical); END_IF
    arrStates[Index].nRequestAssertionID := TO_UDINT(fbJson.GetInt(jsonParam));

    //Set to True to indicate this state has been initialized
    arrStates[Index].bBeamParamsLoaded := bHasAllParameters;

    //Read additional Non-BP Parameters
    bHasAllParameters R= NOT fbJson.HasMember(jsonValue, 'reactive_temp');
    jsonParam := fbJson.FindMember(jsonValue, 'reactive_temp');
    IF (NOT bHasAllParameters) THEN fbLogger(sMsg:= 'Error Loading Temperature Threshold', eSevr:=TcEventSeverity.Critical); END_IF
    arrStates[Index].stReactiveParams.nTempSP := TO_REAL(fbJson.GetString(jsonParam));

    bHasAllParameters R= NOT fbJson.HasMember(jsonValue, 'reactive_pressure');
    jsonParam := fbJson.FindMember(jsonValue, 'reactive_pressure');
    IF (NOT bHasAllParameters) THEN fbLogger(sMsg:= 'Error Loading Pressure Threshold', eSevr:=TcEventSeverity.Critical); END_IF
    arrStates[Index].stReactiveParams.nPressSP := TO_REAL(fbJson.GetString(jsonParam));
END_IF

IF NOT(	bHasAllParameters) THEN
    nErrId := 900+Step;
    bError := TRUE;
    sErrMsg:= CONCAT('Error loading BP Data - Device-State: ',sStateName);
    fbLogger(sMsg:= sErrMsg, eSevr:=TcEventSeverity.Critical);
END_IF

M_LoadSafeBP:=bHasAllParameters;



//TODO
//ADD the rest of the BP
END_METHOD

END_FUNCTION_BLOCK

// MajorComponents/FastFaults/FB_HardwareFFOutput
{attribute 'reflection'}
{attribute 'no_check'}
FUNCTION_BLOCK FB_HardwareFFOutput
VAR CONSTANT
    FF_ARRAY_UPPER_BOUND : UINT := PMPS_PARAM.MAX_FAST_FAULTS;
END_VAR
VAR_INPUT
    {attribute 'pytmc' := '
        pv: ClearFault
        io: o
        field: DESC Might be overidden by PLC writes
     '}
    i_xReset    :    BOOL;
    {attribute 'pytmc' := '
        pv: EnableVeto
        io: o
     '}
    i_xVeto    :    BOOL;
    bAutoReset : BOOL := FALSE; // Set true for the FFO to automatically permit beam again after all fast faults are cleared
    i_sNetID : T_AmsNetID:=''; //Set to the Arbiter AmsNetID to be used for the synchronisation. An empty string means the system will sue local time
END_VAR
VAR_OUTPUT
    {attribute 'pytmc' := '
        pv: FaultHWO
        io: i
        field: DESC Hardware Output Status
     '}
    q_xFastFaultOut    AT %Q*    :    BOOL;
    q_xValidSyncTime : BOOL;// system time bValid output True when sync is successful
END_VAR
VAR_IN_OUT

END_VAR
VAR
    {attribute 'pytmc' := '
        pv: FF
     '}
    astFF : ARRAY[1..FF_ARRAY_UPPER_BOUND] OF ST_FF;

    {attribute 'pytmc' := '
        pv: RegistrationFailure
        io: io
     '}
    xFastFaultRegFail  :   BOOL := FALSE; // Set true if a fast fault fails to register. Holds beam off.
    tFFRegFail : F_TRIG;

    {attribute 'instance-path'}
    {attribute 'noinit'}
    sPath    :    T_MaxString;

    {attribute 'pytmc' := '
        pv: OK
        io: i
     '}
    xOK    :    BOOL:= TRUE; // Current internal state of FFO, indicates if FFO will accept a reset

    rtReset    :    R_TRIG;
    rtResetandOK : R_TRIG;

    nIndex    :    UINT := 1;

    IdxOK: BOOL;

    fbTime : FB_LocalSystemTime := ( bEnable := TRUE, dwCycle := 1 ); //Get current system time, used for override
    fbTime_to_UTC: FB_TzSpecificLocalTimeToSystemTime;
    fbGetTimeZone: FB_GetTimeZoneInformation;
    fbJson : FB_JsonSaxWriter;
    pmpsTypeCode : UDINT := 0; // shows up in json as pmps_typecode
    fbLogger : FB_LogMessage := (
        eSevr := TcEventSeverity.Critical,
        eSubsystem := E_Subsystem.MPS,
        nMinTimeViolationAcceptable := PMPS_PARAM.MAX_FAST_FAULTS);

END_VAR

// <TODO> latch off beam if DI card status goes bad

ACTION EvaluateOutput:

////////////////////////////////////////////////////////////////
// Critical code. Do not touch unless you know what you're doing
////////////////////////////////////////////////////////////////

//<TODO> add diagnostic for success or failure of reset
rtReset(CLK:=i_xReset);
rtResetandOK(CLK:=(rtReset.Q OR bAutoReset) AND xOK);

q_xFastFaultOut S= rtResetandOK.Q;
q_xFastFaultOut R= (NOT xOK OR xFastFaultRegFail);

//Reset OK for next cycle
xOK := True;

////////////////////////////////////////////////////////////////
END_ACTION

{attribute 'no_check'}
METHOD EvaluateOverrides : BOOL
VAR_INPUT
END_VAR
VAR
    FF : REFERENCE TO ST_FF;
    EvalIdx: DINT := 1;
END_VAR
VAR CONSTANT
    MaxTime : DINT:= 4294080;(*49.7 days*)
END_VAR
//Get local System Time
fbTime(sNetID:=i_sNetID);
//Get Time Zone
fbGetTimeZone(sNetID:=i_sNetID,bExecute:=TRUE,tTimeout:=T#10S);
//change local time to UTC to be compatible with unix time epoch widget
fbTime_to_UTC(in:= fbTime.systemTime , tzInfo:=fbGetTimeZone.tzInfo);
q_xValidSyncTime := fbTime.bValid AND NOT fbGetTimeZone.bError;

FOR EvalIdx := 1 TO FF_ARRAY_UPPER_BOUND DO

    FF REF= astFF[EvalIdx];

    IF NOT FF.Info.InUse THEN
        CONTINUE;
    ELSE
        // Veto timer
        IF FF.Ovrd.Deactivate THEN
            FF.Ovrd.Timer.PT := T#0s; // Only needs to be set zero for one cycle
        ELSIF FF.Ovrd.Activate THEN
            FF.Ovrd.StartDT:= TO_DINT(TO_DT(SystemTime_TO_DT(fbTime_to_UTC.out)));
            IF (FF.Ovrd.StartDT < FF.Ovrd.Expiration) THEN
                FF.Ovrd.Expiration:= LIMIT(0,FF.Ovrd.Expiration, FF.Ovrd.StartDT+MaxTime );
                   FF.Ovrd.Timer.PT := TO_DT(FF.Ovrd.Expiration)- SystemTime_TO_DT(fbTime_to_UTC.out);
            END_IF
        END_IF

        // UDINT conversions for ESS module compatibility.
        FF.Ovrd.Timer(
            IN := FF.Ovrd.Activate, // Rising edge activated
            Q => FF.Ovrd.Active);

        FF.Ovrd.tOvrdActivate(CLK:=FF.Ovrd.Active);
        FF.Ovrd.OvrdActLogAck S= FF.Ovrd.tOvrdActivate.Q;

        FF.Ovrd.tOvrdExpiring(CLK:=FF.Ovrd.Active);
        FF.Ovrd.OvrdExpLogAck S= FF.Ovrd.tOvrdExpiring.Q;

        FF.Ovrd.ElapsedTime := TIME_TO_UDINT(FF.Ovrd.Timer.ET);

        FF.Ovrd.RemainingTime := MAX(0, TO_DINT(FF.Ovrd.Timer.PT) - FF.Ovrd.ElapsedTime);

        // Clear pushbuttons
        FF.Ovrd.Activate := FALSE;
        FF.Ovrd.Deactivate := FALSE;

    END_IF
END_FOR
END_METHOD

{attribute 'obsolete' := 'Use EvaluateOverrides instead.'}
METHOD EvaluateVetos : BOOL
VAR_INPUT
END_VAR
END_METHOD

ACTION Execute:
EvaluateOverrides();
EvaluateOutput();
ExecuteLogging();
END_ACTION

{attribute 'no_check'}
METHOD ExecuteLogging : BOOL
VAR_INPUT
END_VAR
VAR
    FF : REFERENCE TO ST_FF;
    logIdx : DINT := 1;
END_VAR
VAR_INST
    HelloTimer : TOF := ( PT:=T#24h );
END_VAR

FOR logIdx := 1 to FF_ARRAY_UPPER_BOUND do

    FF REF= astFF[logIdx];

    IF NOT FF.Info.InUse THEN
        CONTINUE;
    ELSE
        IF FF.FaultAck THEN

            pmpsTypeCode := 1;
            FormulateLogJson(FF);
            fbLogger(sMsg := 'Fault, beam off', eSevr:=TcEventSeverity.Critical);

            FF.FaultAck := FALSE;
        END_IF

        IF FF.Ovrd.OvrdActLogAck THEN

            pmpsTypeCode := 2;
            FormulateLogJson(FF);

            fbLogger(sMsg := 'Override activated', eSevr:=TcEventSeverity.Warning);

            FF.Ovrd.OvrdActLogAck := FALSE;
        END_IF

        IF FF.Ovrd.OvrdExpLogAck THEN

            pmpsTypeCode := 3;
            FormulateLogJson(FF);

            fbLogger(sMsg := 'Override released', eSevr:=TcEventSeverity.Warning);

            FF.Ovrd.OvrdExpLogAck := FALSE;
        END_IF

        IF FF.ClearAck THEN

            pmpsTypeCode := 8;
            FormulateLogJson(FF);

            fbLogger(sMsg := 'Fault cleared', eSevr:=TcEventSeverity.Info);

            FF.ClearAck := FALSE;
        END_IF


    END_IF
END_FOR

// Log registration fault cleared
tFFRegFail(CLK:=xFastFaultRegFail);
IF tFFRegFail.Q THEN
    fbJson.StartObject();
    fbJson.AddKey('pmps_typecode');
    fbJson.AddUdint(5);
    fbJson.AddKey('pmps_path');
    fbJson.AddString(sPath);
    fbJson.EndObject();
    fbJson.CopyDocument(pDoc:=fbLogger.sJson, SIZEOF(fbLogger.sJson));
    fbLogger(sMsg := 'Fast fault registration failure cleared. This may be bad as a fast fault could go unoticed.',
        eSevr:=TcEventSeverity.Warning);
END_IF

// Say hello
HelloTimer.IN := NOT HelloTimer.Q;
HelloTimer();
IF HelloTimer.IN THEN
    pmpsTypeCode := 10;
    FormulateLogJson(FF);
    fbLogger(eSubsystem:=E_Subsystem.NILVALUE,
        eSevr := TcEventSeverity.Info,
        sMsg := 'FFO is alive');
    fbLogger.eSubsystem := E_Subsystem.MPS;
END_IF
END_METHOD

ACTION ExecuteNoLog:
EvaluateOverrides();
EvaluateOutput();
//ExecuteLogging();
END_ACTION

METHOD INTERNAL FormulateLogJson : STRING
VAR_INPUT
    FF : ST_FF;
END_VAR
fbJson.StartObject();
fbJson.AddKey('pmps_typecode');
fbJson.AddUdint(pmpsTypeCode);
fbJson.AddKey('pmps_path');
fbJson.AddString(FF.Info.sPath);
fbJson.AddKey('pmps_device_name');
fbJson.AddString(FF.Info.DevName);
fbJson.EndObject();
fbLogger.sJson := fbJson.GetDocument();
fbJson.ResetDocument();
END_METHOD

{attribute 'no_check'}
METHOD INTERNAL IdxCheckIn : BOOL
VAR_INPUT
    Idx : DINT;
    OK : BOOL;
    Reset : BOOL;
END_VAR
VAR
    stFF : ST_FF;
    BeamPermitted : BOOL;
END_VAR
Idx := LIMIT(1,Idx,FF_ARRAY_UPPER_BOUND);
stFF := THIS^.astFF[Idx];

// Updating internal fault state
stFF.OK := OK;

// Reset and latching logic
stFF.rtReset(CLK:=stFF.Reset (*epics*) OR Reset (*from other PLC logic *) );
stFF.Reset R= stFF.rtReset.Q;
stFF.bsFF(SET := stFF.rtReset.Q OR stFF.Info.AutoReset, RESET1:= NOT OK);

BeamPermitted := stFF.bsFF.Q1 OR stFF.Ovrd.Active OR (i_xVeto AND stFF.Info.Vetoable);

// Fault generation
IF NOT BeamPermitted THEN
    THIS^.xOK := FALSE; //Very clever, thanks Zach!
END_IF

// Fast fault accumulation
stFF.ftCountFault(CLK:=stFF.bsFF.Q1);
IF stFF.ftCountFault.Q THEN PMPS_GVL.AccumulatedFF := PMPS_GVL.AccumulatedFF + 1; END_IF

//Clear pushbuttons
stFF.Reset := FALSE;

// Log when this fault faults
stFF.FaultAck S= stFF.BeamPermitted AND NOT BeamPermitted;

// Log when this fault has cleared
stFF.ClearAck S= BeamPermitted AND NOT stFF.BeamPermitted;

stFF.BeamPermitted := BeamPermitted;

// Copy state back to ff struct
THIS^.astFF[Idx] := stFF;
END_METHOD

{attribute 'no_check'}
METHOD INTERNAL Register : BOOL
VAR_INPUT
    stFFInfo : ST_FFInfo := (
        sPath := '',
        Desc := '',
        TypeCode := 16#00,
        DevName := ''); // Fast fault information

END_VAR
VAR_OUTPUT
    FFOName : T_MaxString;
    Idx : UINT;
END_VAR
VAR
END_VAR
FFOName := THIS^.sPath;
Idx := THIS^.nIndex;

IF THIS^.nIndex <= FF_ARRAY_UPPER_BOUND THEN

    THIS^.astFF[MIN(THIS^.nIndex,FF_ARRAY_UPPER_BOUND)].Info:=stFFInfo;

    THIS^.nIndex := THIS^.nIndex + 1;

    Register := TRUE; // Add successful
ELSE
    fbJson.StartObject();
    fbJson.AddKey('pmps_typecode');
    fbJson.AddUdint(4);
    fbJson.AddKey('pmps_path');
    fbJson.AddString(stFFInfo.sPath);
    fbJson.AddKey('pmps_device_name');
    fbJson.AddString(stFFInfo.DevName);
    fbJson.EndObject();
    fbLogger.sJson := fbJson.GetDocument();
    fbJson.ResetDocument();
    fbLogger(sMsg:='Fast fault registration failed. Too many fast faults on this FFO.',
        eSevr:=TcEventSeverity.Warning,
        eSubsystem:=E_Subsystem.MPS);
    xFastFaultRegFail := TRUE;
    Register := FALSE; // Failed to add name to list
END_IF
END_METHOD

END_FUNCTION_BLOCK

// MajorComponents/FastFaults/FB_FastFault
(* Fast Fault
2019-9-13 A. Wallace

Use this block to generate a beam-off fault. Connects to a fast fault hardware output
function block to contribute to the state of the fast fault output (FFO).

If the i_xOK goes false, the associated FFO will go false, despite the state of any other
contributing fast faults, unless the FFO is currently vetoed.

*)
{attribute 'reflection'}
FUNCTION_BLOCK FB_FastFault
VAR_INPUT

    i_xOK        :    BOOL; // Connect to fast-fault condition (false produces fault)
    i_xReset    :    BOOL; // Resets when i_xOK is true and this is true
    i_xAutoReset : BOOL := FALSE; // Automatically clear fast fault (latching vs non-latching)
    i_xVetoable : BOOL := TRUE; // Mask this fast fault if the FFO veto device is true

    i_DevName : T_MaxString := ''; // Device name for diagnostic
    i_Desc : T_MaxString := ''; // Description of fast fault (you should set at init)
    i_TypeCode : UINT; // Error code for classifying fast faults
END_VAR
VAR_OUTPUT
    o_xFFLine    :    BOOL; //Connect to HW output or another FF input if you like (Optional)
END_VAR
VAR_IN_OUT
    io_fbFFHWO        :    FB_HardwareFFOutput; //Point to FB_HardwareFFOutput of your choice
END_VAR
VAR
    {attribute 'instance-path'}
    {attribute 'noinit'}
    sPath    :    T_MaxString;

    FFInfo : ST_FFInfo;

    RegistrationIdx : UINT := 1; // The index this FF was registered in the FFO

    xInit    :    BOOL :=TRUE;

    InfoStringFmtr : FB_FormatString;

    InUse : T_MaxString;
    AutoReset : T_MaxString;

END_VAR

IF xInit    THEN
    FFInfo.sPath := sPath;
    FFInfo.InUse := True;
    FFInfo.TypeCode := i_TypeCode;
    FFInfo.DevName := i_DevName;
    FFInfo.Desc := i_Desc;
    FFInfo.AutoReset := i_xAutoReset;
    FFInfo.Vetoable := i_xVetoable;

    InUse := BOOL_TO_STRING(FFInfo.InUse);
    AutoReset := BOOL_TO_STRING(FFInfo.AutoReset);
    InfoStringFmtr(sFormat:='%s;%s;%X;%s;%s;%s;',
        arg1 := F_STRING(FFinfo.sPath),
        arg2 := F_STRING(InUse),
        arg3 := F_WORD(FFInfo.TypeCode),
        arg4 := F_STRING(FFInfo.DevName),
        arg5 := F_STRING(FFInfo.Desc),
        arg6 := F_STRING(AutoReset),
        sOut=>FFInfo.InfoString);
    io_fbFFHWO.Register(
        stFFInfo:=FFInfo,
        Idx=>RegistrationIdx);
    //<TODO> if registration doesn't succeed, send warning to diagnostic
    xInit := FALSE;
END_IF

io_fbFFHWO.IdxCheckIn(Idx:=RegistrationIdx, OK := i_xOK, Reset:= i_xReset);

END_FUNCTION_BLOCK

// AncillaryComponents/FB_JsonFileToJsonDoc
FUNCTION_BLOCK FB_JsonFileToJsonDoc
VAR_INPUT
    bExecute             : BOOL; //Rising Edge
    sPLCName			 : STRING;
    sSrcNetId            : T_AmsNetId;
    sSrcPathName         : T_MaxString;
END_VAR
VAR_OUTPUT
    PMPS_jsonDoc 		: SJsonValue;
    bHasPLC              : BOOL;
    bBusy                : BOOL;
    bError               : BOOL;
    nErrId               : UDINT;
    sErrMsg				 :STRING;
END_VAR
VAR_IN_OUT
    io_fbFFHWO    :    FB_HardwareFFOutput;
END_VAR
VAR
    (*Get AMS Net ID*)
    fb_GetLocalAmsNetId: FB_GetLocalAmsNetId;

    (* JSON *)
    fbJson 			: FB_JsonDomParser;
    jsonDoc 		: SJsonValue;
    jsonProp		: SJsonValue;

    (*File*)
    fbFileOpen           : FB_FileOpen;
    fbFileClose          : FB_FileClose;
    fbFileRead           : FB_FileRead;
    hSrcFile             : UINT := 0;(* File handle of the source file *)
    Step: INT;
    index: DINT;
    RisingEdge           : R_TRIG;
    (* Buffer *)
    sbuffRead			:STRING(100000);
    cbReadLength         : UDINT := 0;
    nFileLength	 : UDINT := 0;
    bfbJsonExceptionRaised: BOOL;
    tTimeOut             : TIME := DEFAULT_ADS_TIMEOUT;
    bInit : BOOL;
    (*Logger*)
    tNewMessage : R_TRIG;
    fbLogger : FB_LogMessage := (eSubsystem:=E_SubSystem.MPS, nMinTimeViolationAcceptable:=10);
    (*FFO*)
    FFO    :    FB_FastFault :=(
        i_Desc := 'Fault occurs when there is an error reading json file',
        i_TypeCode := 16#FF13);
END_VAR

(* Get Local AMS net ID*)
IF NOT (bInit) THEN
    fb_GetLocalAmsNetId.bExecute := TRUE;
    bInit :=  TRUE;
END_IF
fb_GetLocalAmsNetId(bExecute:=);

(* Retrieve JSON content *)
RisingEdge(CLK:=bExecute);
CASE Step OF
    0:     (* Idle state *)
          IF RisingEdge.Q THEN
               bBusy := TRUE;
               bError:= FALSE;
               nErrId:=0;
               Step := 1;
               cbReadLength:=0;
               hSrcFile:=0;
               fbLogger(sMsg:='Start Reading Json File.', eSevr:=TcEventSeverity.Info);
               //Clear all json values and read buffer;
               PMPS_jsonDoc := 0;
               jsonDoc:=0;
               jsonProp:=0;
               FOR index:=1  TO 100000 DO
                  sbuffRead[index]:=0;   //clear buffer
               END_FOR
               sErrMsg:='';
               nFileLength:=0;
               jsonDoc := fbJson.ParseDocument(sbuffRead);

          END_IF
    1: (* Open source file *)
           sSrcNetId := fb_GetLocalAmsNetId.AddrString;
          fbFileOpen( bExecute := FALSE );
          fbFileOpen( sNetId := sSrcNetId, sPathName := sSrcPathName,
                         nMode := FOPEN_MODEREAD OR FOPEN_MODETEXT,
                         ePath := PATH_GENERIC, tTimeout := tTimeOut, bExecute := TRUE );
          Step := Step + 1;

    2: (* Check Open file was successful*)
          fbFileOpen( bExecute := FALSE );
          IF NOT fbFileOpen.bBusy THEN
               IF fbFileOpen.bError THEN
                    nErrId := fbFileOpen.nErrId;
                    bError := TRUE;
                    sErrMsg:= CONCAT('Error Opening Json File. E:', TO_STRING(nErrId));
                    Step := 900 + Step;
               ELSE
                    hSrcFile := fbFileOpen.hFile;
                    Step := Step + 1;
               END_IF
          END_IF

    3: (* Read data from source file to buffer string*)
          cbReadLength := 0;
          fbFileRead( bExecute:= FALSE );
          fbFileRead( sNetId:=sSrcNetId, hFile:=hSrcFile,
                         pReadBuff:= ADR(sbuffRead), cbReadLen:= SIZEOF(sbuffRead),
                         bExecute:=TRUE, tTimeout:=tTimeOut );
          Step := Step + 1;

    4: (* Check read file was successful and data read in buffer string*)
         fbFileRead( bExecute:= FALSE );
          IF NOT fbFileRead.bBusy THEN
               IF fbFileRead.bError THEN
                    nErrId := fbFileRead.nErrId;
                    bError := TRUE;
                    sErrMsg:= CONCAT('Error reading Json File. E: ', TO_STRING(nErrId));
                    Step := 900 +Step;
               ELSE
                    cbReadLength := fbFileRead.cbRead;
                    nFileLength := nFileLength + cbReadLength;
                    Step := Step + 1 ;
               END_IF
          END_IF

     5: (* Check Bytes read*)
         IF( nFileLength =0) THEN // oh no, we read zero bytes
            nErrId := fbFileRead.nErrId;
            bError := TRUE;
            sErrMsg:= CONCAT( 'Zero bytes were read from the Json File. E:', TO_STRING(nErrId));
            Step := 900 +Step;
        ELSE // we read something, lets log about it
            fbLogger(sMsg:=CONCAT('Total numbers of Bytes read from file : ', TO_STRING(nFileLength)), eSevr:=TcEventSeverity.Info);
            Step := Step + 1 ;
       END_IF;




     6: (* Close source file *)
        fbFileClose( bExecute := FALSE );
        fbFileClose( sNetId:=sSrcNetId, hFile:=hSrcFile, bExecute:=TRUE, tTimeout:=tTimeOut );
          Step := Step + 1;

     7 :  (*Check file was closed successfully.*)
        fbFileClose( bExecute := FALSE );
          IF NOT fbFileClose.bBusy THEN
               IF fbFileClose.bError THEN
                    nErrId := fbFileClose.nErrId;
                    bError := TRUE;
                    Step:=900+Step;
                    sErrMsg:= CONCAT('Error closing Json File. E:', TO_STRING(nErrId));
               END_IF
               Step := Step + 1;
               hSrcFile := 0;
          END_IF

      8: (* Error or ready => Cleanup *)
          IF (hSrcFile <> 0 ) THEN
               Step := 6; (* Close the source file *)
          ELSE
              (* Ready *)
               Step := 10;
          END_IF

     10: (*Parse read buffer string to JSON DOM object*)
         //cbJsonParserLength := fbJson.CopyDocument(sbuffRead,cbReadLength);
        jsonDoc := fbJson.ParseDocument(sbuffRead);
        bfbJsonExceptionRaised:= fbJson.ExceptionRaised();
        IF (jsonDoc <> 0) AND NOT (bfbJsonExceptionRaised) THEN
            Step := 20;
        ELSE
            Step := 900 + Step;
            nErrId := Step;
            bError := TRUE;
            sErrMsg:= CONCAT('Error Parsing JSON Data. S:',TO_STRING(nErrId));
        END_IF


     20: (*Find the PLC Name*)
        bHasPLC := fbJson.HasMember(jsonDoc, sPLCName);
        IF (bHasPLC) THEN
            jsonProp := fbJson.FindMember(jsonDoc, sPLCName);
            IF jsonProp <> 0 THEN
                Step := Step+1;
                ELSE
                    Step := 900 + Step;
                    nErrId := Step;
                    bError := TRUE;
                    sErrMsg:=  CONCAT('Error Loading PLC data from Json File : ',sPLCName);
                END_IF
        ELSE
            Step := 900 + Step;
            nErrId := Step;
            bError := TRUE;
            sErrMsg:=  CONCAT('Error PLC name not found in Json File : ',sPLCName);
        END_IF

    21: (*write to the PMPS JSonDoc variable*)
      PMPS_jsonDoc := jsonProp;
      Step := 30;

    30: (*ALL good here*)
        fbLogger(sMsg:='Reading and Parsing Json File Completed Successfully.', eSevr:=TcEventSeverity.Info);
         // Release allocated memory
        //jsonDoc := fbJson.NewDocument();
        bExecute:= FALSE;
        bBusy:=FALSE;
        FFO.i_xOK := TRUE;
        Step := 0;

END_CASE

//Fault in error state
IF(Step>=900) THEN
    FFO.i_xOK := FALSE;
    bBusy:=FALSE;
    Step:=0;
END_IF
ACT_FFO();
ACT_LOGGER();

ACTION ACT_FFO:
(*FAST FAULT*)
FFO(i_xOK := ,
    i_xReset := ,
    i_xAutoReset :=TRUE,
    i_DevName := sPLCName,
    io_fbFFHWO := io_fbFFHWO);
END_ACTION

ACTION ACT_Logger:
// Log valve open
tNewMessage(CLK:= NOT(FbLogger.sMsg = sErrMsg) AND NOT (sErrMsg =''));
IF tNewMessage.Q THEN fbLogger(sMsg:= sErrMsg, eSevr:=TcEventSeverity.Critical); END_IF
END_ACTION

END_FUNCTION_BLOCK

// AncillaryComponents/FB_PressSensor_FFO
FUNCTION_BLOCK FB_PressSensor_FFO
VAR_INPUT
    {attribute 'pytmc' := '
        pv: Press
        io: input
        field: EGU Torr
        field: PREC 2
    '}
    rPress : REAL;
    {attribute 'pytmc' := '
        pv: FAULT_SP
        io: input
        field: EGU Torr
        field: PREC 2
    '}
    fFaultThreshold : LREAL; //Faults when the threshold is reached. Trigger value.
    {attribute 'pytmc' := '
        pv: FAULT_SP_HYS
        io: input
        field: EGU %
        field: PREC 2
    '}
    fHysteresis : LREAL :=1; // percentage determining how far below the trigger value the fault should be released
    sDevName: STRING;
    bVeto : BOOL:=FALSE; // This Fault will be will not trip the beam if the bVeto is TRUE
    bAutoReset : BOOL:=TRUE;
END_VAR
VAR_IN_OUT
    io_fbFFHWO    :    FB_HardwareFFOutput;
END_VAR
VAR_OUTPUT
END_VAR
VAR
    {attribute 'instance-path'}
    {attribute 'noinit'}
    sPath: STRING;
    bFAULT_OK:BOOL :=FALSE;
    FFO    :    FB_FastFault :=(
        i_Desc := 'Fault occurs when the temprature trip point is reached',
        i_TypeCode := 16#f700);
    rtRESET	:	R_TRIG;
    ftFAULT	:	F_TRIG;
    fbLogger : FB_LogMessage := (eSubsystem:=E_SubSystem.MPS, nMinTimeViolationAcceptable:=10);
END_VAR


//Verify Hysteresis is between 1-100, Shouldn't be 0. shouldn't be a 100 either.
fHysteresis:=  LIMIT(1, fHysteresis, 100);

// Evaluate the threshold trip point
IF (rPress >= fFaultThreshold) THEN
    bFAULT_OK := FALSE;
ELSIF (rPress < (fFaultThreshold - fFaultThreshold*fHysteresis/100)) THEN
    bFAULT_OK := TRUE;
END_IF



ACT_Logger();

(*FAST FAULT*)
FFO(i_xOK := bFAULT_OK OR bVeto,
    i_xReset :=,
    i_xAutoReset := bAutoReset,
    i_DevName := sDevName,
    io_fbFFHWO := io_fbFFHWO);

ACTION ACT_Logger:
ftFAULT(CLK:= FFO.i_xOK);
rtRESET(CLK:=FFO.i_xOK);

IF(ftFAULT.Q) THEN
    fbLogger(sMsg := 'Temp Threshold Fault, beam off', eSevr:=TcEventSeverity.Critical);
END_IF

IF(rtRESET.Q) THEN
    fbLogger(sMsg := 'Temp Threshold Fault condition clear', eSevr:=TcEventSeverity.Info);
END_IF
END_ACTION

END_FUNCTION_BLOCK

// AncillaryComponents/FB_TempSensor_FFO
FUNCTION_BLOCK FB_TempSensor_FFO EXTENDS FB_TempSensor
VAR_INPUT
    {attribute 'pytmc' := '
        pv: FAULT_SP
        io: input
        field: EGU C
        field: PREC 2
    '}
    fFaultThreshold : LREAL; //Faults when the threshold is reached. Trigger value.
    {attribute 'pytmc' := '
        pv: FAULT_SP_HYS
        io: input
        field: EGU %
        field: PREC 2
    '}
    fHysteresis : LREAL :=1; // percentage determining how far below the trigger value the fault should be released
    sDevName: STRING;
    bVeto : BOOL:=FALSE; // This Fault will be will not trip the beam if the bVeto is TRUE
    bAutoReset : BOOL:=TRUE;
END_VAR
VAR_IN_OUT
    io_fbFFHWO    :    FB_HardwareFFOutput;
END_VAR
VAR_OUTPUT
END_VAR
VAR
    {attribute 'instance-path'}
    {attribute 'noinit'}
    sPath: STRING;
    bFAULT_OK:BOOL :=FALSE;
    FFO    :    FB_FastFault :=(
        i_Desc := 'Fault occurs when the temprature trip point is reached',
        i_TypeCode := 16#f700);
    rtRESET	:	R_TRIG;
    ftFAULT	:	F_TRIG;
    ftConnected	:	F_TRIG;
    fbLogger : FB_LogMessage := (eSubsystem:=E_SubSystem.MPS, nMinTimeViolationAcceptable:=10);
END_VAR

 // The manual states that we are disconnected if we are both overrange and in an error state
bConnected := NOT (bOverrange AND bError);
fTemp := INT_TO_LREAL(iRaw) * fResolution;

//Verify Hysteresis is between 1-100, Shouldn't be 0. shouldn't be a 100 either.
fHysteresis:=  LIMIT(1, fHysteresis, 100);

// Evaluate the threshold trip point
IF (fTemp >= fFaultThreshold) THEN
    bFAULT_OK := FALSE;
ELSIF (fTemp < (fFaultThreshold - fFaultThreshold*fHysteresis/100)) THEN
    bFAULT_OK := TRUE;
END_IF
bFAULT_OK R= NOT bConnected;


ACT_Logger();

(*FAST FAULT*)
FFO(i_xOK := bFAULT_OK OR bVeto,
    i_xReset :=,
    i_xAutoReset := bAutoReset,
    i_DevName := sDevName,
    io_fbFFHWO := io_fbFFHWO);

ACTION ACT_Logger:
ftFAULT(CLK:= FFO.i_xOK);
rtRESET(CLK:=FFO.i_xOK);
ftConnected(CLK:= bConnected);

IF(ftConnected.Q) THEN
    fbLogger(sMsg := 'Sensor Connection Fault, beam off', eSevr:=TcEventSeverity.Critical);
END_IF

IF(ftFAULT.Q) THEN
    fbLogger(sMsg := 'Temp Threshold Fault, beam off', eSevr:=TcEventSeverity.Critical);
END_IF

IF(rtRESET.Q) THEN
    fbLogger(sMsg := 'Temp Threshold Fault condition clear', eSevr:=TcEventSeverity.Info);
END_IF
END_ACTION

END_FUNCTION_BLOCK

// HelperFunctions/TypeTranslators/APT_TO_IO
FUNCTION APT_TO_IO : ST_PMPS_Aperture_IO
VAR_INPUT
    Apt : ST_PMPS_Aperture;
END_VAR
VAR
END_VAR

APT_TO_IO.Height := Apt.Height;
APT_TO_IO.Width := Apt.Width;
APT_TO_IO.xOK := Apt.xOK;

END_FUNCTION

// HelperFunctions/TypeTranslators/ATT_TO_IO
FUNCTION ATT_TO_IO : ST_PMPS_Attenuator_IO
VAR_INPUT
    Att : ST_PMPS_Attenuator;
END_VAR
VAR
END_VAR

ATT_TO_IO.nTran := Att.nTran;
ATT_TO_IO.xAttOK := Att.xAttOK;

END_FUNCTION

// HelperFunctions/TypeTranslators/BP_TO_IO
{attribute 'no_check'}
FUNCTION BP_TO_IO : ST_BeamParams_IO
VAR_INPUT
    BP : ST_BeamParams;
END_VAR
VAR
    idx : UINT := 0;
END_VAR


FOR idx := 1 TO PMPS_GVL.AUX_ATTENUATORS DO
    BP_TO_IO.astAttenuators[idx] := ATT_TO_IO(BP.astAttenuators[idx]);
END_FOR

FOR idx := 1 TO PMPS_GVL.MAX_APERTURES DO
    BP_TO_IO.astApertures[idx] := APT_TO_IO(BP.astApertures[idx]);
END_FOR

BP_TO_IO.aVetoDevices := BP.aVetoDevices;
BP_TO_IO.nTran := BP.nTran;
BP_TO_IO.nCohortInt := ULINT_TO_UDINT(BP.nCohortInt);
BP_TO_IO.neVRange := BP.neVRange;
BP_TO_IO.neV := BP.neV;
BP_TO_IO.nBCRange := BP.nBCRange;
BP_TO_IO.nBeamClass := BP.nBeamClass;
BP_TO_IO.nMachineMode := BP.nMachineMode;
BP_TO_IO.nRate := BP.nRate;
BP_TO_IO.xValid := BP.xValid;
BP_TO_IO.xValidToggle := BP.xValidToggle;

END_FUNCTION

// HelperFunctions/TypeTranslators/F_DeviceState_To_DeviceStateExt
FUNCTION F_DeviceState_To_DeviceStateExt : ST_DeviceStateExt
VAR_INPUT
    stDeviceState    :    ST_DeviceState;
    xValid    :    BOOL;
END_VAR
VAR
END_VAR

F_DeviceState_To_DeviceStateExt.nStateRef := stDeviceState.nStateRef;
F_DeviceState_To_DeviceStateExt.rPosition    :=    stDeviceState.rPosition;
F_DeviceState_To_DeviceStateExt.rTolerance    :=    stDeviceState.rTolerance;
F_DeviceState_To_DeviceStateExt.sStateName    := stDeviceState.sStateName;
F_DeviceState_To_DeviceStateExt.stReqBeamParam    := stDeviceState.stReqBeamParam;
F_DeviceState_To_DeviceStateExt.xValid := xValid;

END_FUNCTION

// HelperFunctions/TypeTranslators/IO_TO_APT
FUNCTION IO_TO_APT : ST_PMPS_Aperture
VAR_INPUT
    IO : ST_PMPS_Aperture_IO;
END_VAR
VAR
END_VAR

IO_TO_APT.Height := IO.Height;
IO_TO_APT.Width := IO.Width;
IO_TO_APT.xOK := IO.xOK;

END_FUNCTION

// HelperFunctions/TypeTranslators/IO_TO_ATT
FUNCTION IO_TO_ATT : ST_PMPS_Attenuator
VAR_INPUT
    IO : ST_PMPS_Attenuator_IO;
END_VAR
VAR
END_VAR

IO_TO_ATT.nTran := IO.nTran;
IO_TO_ATT.xAttOK := IO.xAttOK;

END_FUNCTION

// HelperFunctions/TypeTranslators/IO_TO_BP
{attribute 'no_check'}
FUNCTION IO_TO_BP : ST_BeamParams
VAR_INPUT
    IO : ST_BeamParams_IO;
END_VAR
VAR
    idx : UINT;
END_VAR


FOR idx := 1 TO PMPS_GVL.AUX_ATTENUATORS DO
    IO_TO_BP.astAttenuators[idx] := IO_TO_ATT(IO.astAttenuators[idx]);
END_FOR

FOR idx := 1 TO PMPS_GVL.MAX_APERTURES DO
    IO_TO_BP.astApertures[idx] := IO_TO_APT(IO.astApertures[idx]);
END_FOR

IO_TO_BP.aVetoDevices := IO.aVetoDevices;
IO_TO_BP.nTran := IO.nTran;
IO_TO_BP.nCohortInt := ULINT_TO_UDINT(IO.nCohortInt);
IO_TO_BP.neVRange := IO.neVRange;
IO_TO_BP.neV := IO.neV;
IO_TO_BP.nBCRange := IO.nBCRange;
IO_TO_BP.nBeamClass := IO.nBeamClass;
IO_TO_BP.nMachineMode := IO.nMachineMode;
IO_TO_BP.nRate := IO.nRate;
IO_TO_BP.xValid := IO.xValid;
IO_TO_BP.xValidToggle := IO.xValidToggle;

END_FUNCTION

// HelperFunctions/F_AttenuatorOK
(*
Indicates if the attenuator can be considered safe for a device,
given its status word.

In local mode, the atteunator ignores PMPS requests, following a local
setpoint. In this mode, a device cannot trust that the attenuator will not
increase transmission beyond its own setpoint. Therefore any
indication of a changing transmission should cause a fault.

In PMPS mode, if a device has submitted a preemptive request and received
acknowledgement, then the transmission setpoint will be governed at least
by that device's setpoint. Therefore, the attenuator may be moving without
generating a fault.
*)
FUNCTION F_AttenuatorOK : BOOL
VAR_INPUT
    xStatus : WORD;
END_VAR
VAR
END_VAR

IF xStatus.2 THEN // Local mode
    F_AttenuatorOK := xStatus.0 and NOT xStatus.1;
ELSIF xStatus.3 AND NOT xStatus.2 THEN // PMPS mode
    F_AttenuatorOK := TRUE;
END_IF

F_AttenuatorOK := xStatus.4 AND F_AttenuatorOK;

END_FUNCTION

// HelperFunctions/F_BPWithID
FUNCTION F_BPWithID : ST_BP_ArbInternal
VAR_INPUT
    BP : REFERENCE TO ST_BeamParams;
    ID : DWORD;
END_VAR
VAR
    BpInt : ST_BP_ArbInternal;
END_VAR

MEMCPY(ADR(F_BPWithID), ADR(BP), SIZEOF(BP));
F_BPWithID.nId := ID;

END_FUNCTION

// HelperFunctions/F_DifferentBeamParams
(*Compares BeamParam1 to BeamParam2, if any parameters of BeamParam1 are different than BeamParam2
the result will be true. *)
{attribute 'no_check'}
FUNCTION F_DifferentBeamParams : BOOL
VAR_INPUT
    BeamParam1    :    ST_BeamParams;
    BeamParam2    :    ST_BeamParams;
END_VAR
VAR
    xAttOK: BOOL := FALSE;
    xPPmjOK: BOOL := FALSE;
    xEvOK: BOOL := FALSE;
    xRateOK: BOOL := FALSE;
    xaStopper : BOOL := FALSE;
    xaAtt : BOOL := FALSE;
    xaApt : BOOL := FALSE;
    xBCOK : BOOL := FALSE;

    idx : UINT;


END_VAR

xAttOK := BeamParam1.nTran <> BeamParam2.nTran;
xEvOK := BeamParam1.neVRange <> BeamParam2.neVRange;
xRateOK     := BeamParam1.nRate <> BeamParam2.nRate;
xBCOK	:= BeamParam1.nBCRange <> BeamParam2.nBCRange;// OR BeamParam1.nBeamClass <> BeamParam2.nBeamClass ; //Is this right?


//ast Attenuators
FOR idx:=1 TO PMPS_GVL.AUX_ATTENUATORS DO
    xaAtt S= (BeamParam1.astAttenuators[idx].nTran <> BeamParam2.astAttenuators[idx].nTran);
END_FOR

// Stoppers
FOR idx:=1 TO PMPS_GVL.MAX_VETO_DEVICES DO
    xaStopper S= (BeamParam1.aVetoDevices[idx] <> BeamParam2.aVetoDevices[idx]);
END_FOR

// ast Apertures
FOR idx:=1 TO PMPS_GVL.MAX_APERTURES DO
    xaApt S= (BeamParam1.astApertures[idx].Height <> BeamParam2.astApertures[idx].Height) OR
            (BeamParam1.astApertures[idx].Width <> BeamParam2.astApertures[idx].Width);
END_FOR


F_DifferentBeamParams := xAttOK OR xPPmjOK OR xEvOK OR xRateOK OR xaStopper OR xaAtt OR xaApt OR xBCOK;

END_FUNCTION

// HelperFunctions/F_eVExcludeRange
FUNCTION F_eVExcludeRange : DWORD
(*
    Given an lower and upper end of an exclusion range, return the corresponding eV bitmask.

    eVs between fLower and fUpper will be considered unsafe, and eVs outside of this range will be
    considered safe, with the exception of the endpoints and values near the endpoints if they land
    far from an eV boundary.

    Call this in your init cycle to set up your eV bitmasks for more readable code
    that is also more resiliant to eV range definition adjustments.
*)
VAR_INPUT
    fLower: REAL;
    fUpper: REAL;
END_VAR


F_eVExcludeRange := F_eVIncludeRange(0, fLower) OR F_eVIncludeRange(fUpper, PMPS_GVL.g_areVBoundaries[PMPS_GVL.g_cBoundaries]);

END_FUNCTION

// HelperFunctions/F_eVIncludeRange
FUNCTION F_eVIncludeRange : DWORD
(*
    Given an lower and upper end of an inclusion range, return the corresponding eV bitmask.

    eVs between fLower and fUpper will be considered safe, with the exception of the endpoints and values
    near the endpoints if they land far from an eV boundary.

    Call this in your init cycle to set up your eV bitmasks for more readable code
    that is also more resiliant to eV range definition adjustments.
*)
VAR_INPUT
    fLower: REAL;
    fUpper: REAL;
END_VAR
VAR
    nBitmask: DWORD := 0;
    nIndex: INT;
    nBit: USINT := 0;
    fPrev: REAL := 0;
END_VAR


FOR nIndex := 0 TO PMPS_GVL.g_cBoundaries DO
    IF fLower <= fPrev AND fUpper >= PMPS_GVL.g_areVBoundaries[nIndex] THEN
        nBitmask := nBitmask + SHL(1, nBit);
    END_IF
    fPrev := PMPS_GVL.g_areVBoundaries[nIndex];
    nBit := nBit + 1;
END_FOR

F_eVIncludeRange := nBitmask;

END_FUNCTION

// HelperFunctions/F_eVRangeCalculator
(*
A. Wallace 2019-8-8

Provides bit range of eV.

LastWord = 0 (Result)
----------------------------------
reV = 300 = (0000_0000_0000_0010)
reV = 301 = (0000_0000_0000_0100)

LastWord = 0000_0000_0000_0010 (Result)
----------------------------------
reV = 300 + <rHyst = (0000_0000_0000_0110)
reV = 300 + >rHyst = (0000_0000_0000_0100)

*)
{attribute 'no_check'}
FUNCTION F_eVRangeCalculator : DWORD // Bit-range of current photon energy
VAR_INPUT
    reV    :    REAL; // Photon energy (keV)
    LastWord    :    DWORD; // Range word of previous cycle
END_VAR
VAR
    nIndex: INT;
    RangeWord: DWORD;
    rPreviousBoundary: REAL := 0;

    MaxEv    :    REAL := PMPS_GVL.g_areVBoundaries[PMPS_GVL.g_cBoundaries];

    Boundaries : ARRAY [0..PMPS_GVL.g_cBoundaries] OF REAL;
END_VAR

{IF defined (L)}
    Boundaries := PMPS_GVL.g_areVBoundariesL;
{ELSIF defined (K)}
    Boundaries := PMPS_GVL.g_areVBoundariesK;
{END_IF}

MaxEv := Boundaries[PMPS_GVL.g_cBoundaries];

IF reV <= 0 OR reV > MaxEv THEN F_eVRangeCalculator := 16#FFFF_FFFF; RETURN; END_IF // Failsafe

FOR nIndex := 0 TO PMPS_GVL.g_cBoundaries DO

    // If previously active then check if it should be cleared
    IF LastWord.0 THEN
        // Hysteresis condition
        IF (reV > MIN(Boundaries[nIndex] + PMPS_GVL.reVHyst, MaxEv) ) OR
        (reV < MAX(rPreviousBoundary - PMPS_GVL.reVHyst, 0) ) THEN
            RangeWord.0 := 0; // If out of range of hys. mark inactive
        ELSE
            RangeWord.0 := 1;
        END_IF
    ELSE // Check if we should mark as active
        IF (reV <= Boundaries[nIndex]) AND
        (reV > rPreviousBoundary) OR
         (nIndex = 0 AND reV = 0 ) THEN
            RangeWord.0 := 1;
        END_IF
    END_IF

    // Catch if the hysteresis is set too large for the range
    IF rPreviousBoundary + PMPS_GVL.reVHyst >= Boundaries[nIndex] THEN
        RangeWord.0 := 1; // Setting the bit true here as a failsafe
        //<TODO> Add major error or warning here
    END_IF

    rPreviousBoundary := Boundaries[nIndex];
    // Shift to next bit
    RangeWord := ROR(RangeWord, 1);
    LastWord := SHR(LastWord, 1);

END_FOR

F_eVRangeCalculator := RangeWord;

END_FUNCTION

// HelperFunctions/F_eVWithinSpec
//reV must be within permitted range.
{attribute 'no_check'}
FUNCTION F_eVWithinSpec : BOOL
VAR_INPUT
    reV    :    REAL;    //Photon energy to check if within permitted range
    nPermittedRange    :    DWORD; //Permitted range
END_VAR
VAR
    //Holding register for permitted ranges
    nPermittedRangeHolding    :    DWORD;
    //For loop counter
    nIndex    :    INT;
    // Lower boundary for range check
    rPreviousBoundary: REAL := 0;
    Boundaries: ARRAY [0..PMPS_GVL.g_cBoundaries] OF REAL;
END_VAR

(* How this works:
The within range bool is initialized to false.
Load the word representation of ranges into a holding register.
If the bit at position zero of the holding register is true, and the input eV is
below the boundary at the index position of the boundary array, and the previous boundary
(which initializes at 0), then the within range bool is set.
Then, we stash the upper boundary as the lower boundary for the next comparison,
and shift the holding register right, which moves the next bit to the zero position.
*)

{IF defined (L)}
    Boundaries := PMPS_GVL.g_areVBoundariesL;
{ELSIF defined (K)}
    Boundaries := PMPS_GVL.g_areVBoundariesK;
{END_IF}

nPermittedRangeHolding := nPermittedRange;

FOR nIndex := 0 TO PMPS_GVL.g_cBoundaries DO

    F_eVWithinSpec S= nPermittedRangeHolding.0 AND(
        (reV <= Boundaries[nIndex]) AND
        (reV >= rPreviousBoundary) );

    IF F_eVWithinSpec THEN RETURN; END_IF

    rPreviousBoundary := Boundaries[nIndex];
    nPermittedRangeHolding := SHR(nPermittedRangeHolding, 1);
END_FOR

END_FUNCTION

// HelperFunctions/F_InitTestBP
// Establishes a BP set for testing.
// Specifically this means a BP that has all the status bits set to an OK state
FUNCTION F_InitTestBP : ST_BeamParams
VAR_INPUT
    BP : ST_BeamParams;
END_VAR
VAR
END_VAR

END_FUNCTION

// HelperFunctions/F_PMPS_JSON
FUNCTION F_PMPS_JSON : STRING
VAR_INPUT
    sDevName : STRING := '';
    sPath : STRING := '';
    nTypeCode : UINT := 0;
END_VAR
VAR

END_VAR


PMPS_TOOLS.fbJson.StartObject();
PMPS_TOOLS.fbJson.AddKey('pmps_typecode');
PMPS_TOOLS.fbJson.AddUdint(nTypeCode);
PMPS_TOOLS.fbJson.AddKey('pmps_path');
PMPS_TOOLS.fbJson.AddString(sPath);
PMPS_TOOLS.fbJson.AddKey('pmps_device_name');
PMPS_TOOLS.fbJson.AddString(sDevName);
PMPS_TOOLS.fbJson.EndObject();
F_PMPS_JSON := PMPS_TOOLS.fbJson.GetDocument();
PMPS_TOOLS.fbJson.ResetDocument();

END_FUNCTION

// HelperFunctions/F_SafeBPCompare
(*Compares BeamParam1 to BeamParam2: if the parameters of BeamParam1 are more conservative than BeamParam2
the result will be true. *)
// Does not consider status. Status must be evaluated elsewhere.
{attribute 'no_check'}
FUNCTION F_SafeBPCompare : BOOL
VAR_INPUT
    BeamParam1    :    ST_BeamParams; //Must be more conservative than 2
    BeamParam2    :    ST_BeamParams;
END_VAR
VAR
    // Internal Attenuation OK boolean
    xAttOK: BOOL := FALSE;
    // Internal Per-pulse energy OK boolean
    xPPmjOK: BOOL := FALSE;
    // Internal photon energy OK boolean
    xEvOK: BOOL := FALSE;
    // Internal Beam Rate OK boolean
    xRateOK: BOOL;
    //Internal Beam Class Range OK boolean
    xBCOK : BOOL := FALSE;
    idx : UINT;
    xAuxAttOK : BOOL := TRUE;
    xAuxAprtOK : BOOL := TRUE;

    Att1 : REFERENCE TO ST_PMPS_Attenuator;
    Att2 : REFERENCE TO ST_PMPS_Attenuator;

END_VAR


xAttOK := BeamParam1.nTran <= MIN(PMPS_GVL.TRANS_SCALING_FACTOR, (BeamParam2.nTran *(PMPS_GVL.TRANS_SCALING_FACTOR+PMPS_PARAM.TRANS_MARGIN))/PMPS_GVL.TRANS_SCALING_FACTOR );
xEvOK := (BeamParam1.neVRange AND BeamParam2.neVRange) = BeamParam1.neVRange;
xRateOK    := (BeamParam1.nRate <= BeamParam2.nRate) OR (PMPS_GVL.stCurrentBeamParameters.nMachineMode =1); //ignore in SC mode
xBCOK := ((BeamParam1.nBCRange AND BeamParam2.nBCRange) = BeamParam1.nBCRange) OR (PMPS_GVL.stCurrentBeamParameters.nMachineMode =0); //ignore in NC mode;

FOR idx:=1 to PMPS_GVL.AUX_ATTENUATORS DO
    Att1 REF= BeamParam1.astAttenuators[idx];
    Att2 REF= BeamParam2.astAttenuators[idx];
    xAuxAttOK R= ( Att1.nTran > MIN( PMPS_GVL.TRANS_SCALING_FACTOR, ( (Att2.nTran *(PMPS_GVL.TRANS_SCALING_FACTOR+PMPS_PARAM.TRANS_MARGIN))/PMPS_GVL.TRANS_SCALING_FACTOR ) ) );
END_FOR

FOR idx:=1 to PMPS_GVL.MAX_APERTURES DO
    xAuxAprtOK R= BeamParam1.astApertures[idx].Height > BeamParam2.astApertures[idx].Height OR
    BeamParam1.astApertures[idx].Width > BeamParam2.astApertures[idx].Width;
END_FOR

F_SafeBPCompare := xAttOK AND xEvOK AND xRateOK AND xAuxAprtOK AND xAuxAttOK AND xBCOK;

END_FUNCTION

// HelperFunctions/F_SafeBPCompare0Rate
(*Compares BeamParam1 to BeamParam2: if the parameters of BeamParam1 are more conservative than BeamParam2
the result will be true. *)
(* When the Mode PV is in Cu 0-rate means this function will return true regardless of other conditions if the beam rate
is zero *)
(* When the Mode PV is in SC 0-bc means this function will return true regardless of other conditions if the beam class
is zero *)
FUNCTION F_SafeBPCompare0Rate : BOOL
VAR_INPUT
    BeamParam1    :    ST_BeamParams; //Must be more conservative than 2
    BeamParam2    :    ST_BeamParams;
END_VAR
VAR

    // Beam-rate is zero, masks all others considerations.
    xZeroRate: BOOL;
    //Beam class is zero i.e beam off, masks all other considerations.
    xZeroBC : BOOL;

END_VAR


xZeroRate  := (BeamParam1.nRate = 0) AND (PMPS_GVL.stCurrentBeamParameters.nMachineMode = 0);
xZeroBC  := (BeamParam1.nBCRange <= 1) AND (PMPS_GVL.stCurrentBeamParameters.nMachineMode =1);

F_SafeBPCompare0Rate := (xZeroRate OR xZeroBC) OR F_SafeBPCompare(BeamParam1, BeamParam2);

END_FUNCTION

// HelperFunctions/F_SetBeamParams
FUNCTION F_SetBeamParams : ST_BeamParams
VAR_INPUT
    nTran    :    REAL := 0;
    neVRange    :    DWORD := 0;
    nRate    :    UDINT := 0;
    nBCRange : WORD := 0;
    astAuxAtt : ARRAY [1..PMPS_GVL.AUX_ATTENUATORS] OF ST_PMPS_Attenuator;
END_VAR
VAR
    BeamParams    :    ST_BeamParams;

END_VAR

BeamParams.nTran := LIMIT(0,nTran,PMPS_GVL.TRANS_SCALING_FACTOR);
BeamParams.astAttenuators := astAuxAtt;
BeamParams.neVRange := neVRange;
BeamParams.nRate    := MIN(nRate,1000000);
BeamParams.nBCRange	:= MIN(nBCRange,32767);

F_SetBeamParams    := BeamParams;

END_FUNCTION

// HelperFunctions/F_SetGoodAttStatus
//Use for testing purposes to set the attenuator status to a good state
FUNCTION F_SetGoodAttStatus : UINT
VAR_INPUT
    xStatus : UINT;
END_VAR
VAR
END_VAR

xStatus.0 := 1;
xStatus.3 := 1;
xStatus.4 := 1;

END_FUNCTION

// HelperFunctions/F_SetStateParams
FUNCTION F_SetStateParams : BOOL;
VAR_INPUT
    nStateRef    :    UDINT;
    rPosition    :    REAL;
    rTolerance: REAL;
    stBeamParams    :    ST_BeamParams;
END_VAR
VAR_IN_OUT
    Table    :    FB_LinearDeviceStateTable;
END_VAR
VAR
    stDeviceState    :    ST_DeviceState;

END_VAR

stDeviceState.nStateRef := nStateRef;
stDeviceState.rPosition := rPosition;
stDeviceState.rTolerance := rTolerance;
stDeviceState.stReqBeamParam := stBeamParams;

Table.A_Add(
    key := nStateRef,
    putValue := stDeviceState
);

F_SetStateParams := Table.bOk;

END_FUNCTION

// MajorComponents/FB_LinearDeviceStateTable
(* This function block implements simple database. Data element values are stored in the hash table.  *)
{attribute 'no_check'}
FUNCTION_BLOCK FB_LinearDeviceStateTable
VAR_INPUT
    key         : DWORD := 0;(* Entry key: used by A_Lookup, A_Remove method, the key variable is also used by A_Add method *)
    putPosPtr    : POINTER TO T_HashTableEntry := 0;(* Hash table entry position pointer (used by A_Find, A_GetNext, A_GetPrev) *)
    putValue     : ST_DeviceState;(* Hash table entry value (used by A_AddHead, A_AddTail, A_Find )*)
END_VAR
VAR_OUTPUT
    bOk            : BOOL := FALSE;(* TRUE = Success, FALSE = Failed *)
    getPosPtr    : POINTER TO T_HashTableEntry := 0;(* Returned hash table entry position pointer *)
    getValue     : ST_DeviceState;(* Returned hash table entry value *)
    nCount        : UDINT := 0;(* Hash table size (number of used entries, used by A_Count) *)
END_VAR
VAR
    dataPool    : ARRAY[0..PMPS_GVL.MAX_DEVICE_STATES] OF ST_DeviceState;(* Structured data element pool *)
    entries        : ARRAY[0..PMPS_GVL.MAX_DEVICE_STATES] OF T_HashTableEntry;(* Max. number of hash table entries. The value of table entry = 32 bit integer (pointer to dataPool-array-entry) *)
    fbTable     : FB_HashTableCtrl;(* basic hash table control function block *)
    hTable         : T_HHASHTABLE;(* hash table handle *)
    pRefPtr        : POINTER TO ST_DeviceState := 0;
    indexOfElem    : ULINT;(* Integer value (max. size: x86=>32bit, x64=>64bit)*)
END_VAR

;

ACTION A_Add:
(* Adds entry to the table *)
MEMSET( ADR( getValue ), 0, SIZEOF( getValue ) );
getPosPtr := 0;

fbTable.A_Add( hTable := hTable, key := key, putValue := 16#0000_0000(* we will set this value later *), getPosPtr=>getPosPtr, bOk=>bOk );(* Add new element to the table, getPosPtr points to the new entry *)
IF fbTable.bOk THEN(* Success *)
    fbTable.A_GetIndexAtPosPtr( hTable := hTable, putPosPtr := getPosPtr, getValue =>indexOfElem, bOk=>bOk );(* Get array index of getPosPtr entry *)
    IF fbTable.bOk THEN(* Success *)
        pRefPtr     := ADR( dataPool[indexOfElem] );(* Get pointer to the data element *)

        pRefPtr^ := putValue;(* copy application value *)

        fbTable.A_Add( hTable := hTable, key := key, putValue := pRefPtr, bOk=>bOk );(* Assign the entry value = pointer to the data element *)
        IF fbTable.bOk THEN(* Success *)
            getValue := putValue;
        END_IF
    END_IF
END_IF
END_ACTION

ACTION A_Count:
(* Count number of used entries *)
nCount := hTable.nCount;
bOk := TRUE;
END_ACTION

ACTION A_GetFirst:
(* Get first entry position pointer and value *)
MEMSET( ADR( getValue ), 0, SIZEOF( getValue ) );
getPosPtr := 0;

fbTable.A_GetFirst( hTable := hTable, putPosPtr := putPosPtr, getValue=>pRefPtr, getPosPtr=>getPosPtr, bOk=>bOk );
IF fbTable.bOk THEN
    getValue := pRefPtr^;
END_IF
END_ACTION

ACTION A_GetNext:
(* Get next entry position pointer and value *)
MEMSET( ADR( getValue ), 0, SIZEOF( getValue ) );
getPosPtr := 0;
bOk := FALSE;

IF putPosPtr = 0 THEN
    RETURN;
END_IF

fbTable.A_GetNext( hTable := hTable, putPosPtr := putPosPtr, getValue=>pRefPtr, getPosPtr=>getPosPtr, bOk=>bOk );
IF fbTable.bOk THEN
    getValue := pRefPtr^;
END_IF
END_ACTION

ACTION A_Lookup:
(* Lookup for entry by key  *)
MEMSET( ADR( getValue ), 0, SIZEOF( getValue ) );
getPosPtr := 0;

fbTable.A_Lookup( key := key, hTable := hTable, putPosPtr := putPosPtr, getValue=>pRefPtr, getPosPtr=>getPosPtr, bOk=>bOk );
IF fbTable.bOk THEN
    getValue := pRefPtr^;
END_IF
END_ACTION

ACTION A_Remove:
(* Search for entry and remove it *)
MEMSET( ADR( getValue ), 0, SIZEOF( getValue ) );
getPosPtr := 0;

fbTable.A_Remove( key := key, hTable := hTable, putPosPtr := putPosPtr, getValue=>pRefPtr, getPosPtr=>getPosPtr, bOk=>bOk );
IF fbTable.bOk THEN
    getValue := pRefPtr^;
END_IF
END_ACTION

ACTION A_Reset:
(* Reset/initialize linked list *)
MEMSET( ADR( getValue ), 0, SIZEOF( getValue ) );
getPosPtr := 0;
bOk := F_CreateHashTableHnd( ADR( entries ), SIZEOF( entries ), hTable );(* Intialize table handle *)
fbTable.A_Reset( hTable := hTable, bOk=>bOk );
nCount := 0;
END_ACTION

END_FUNCTION_BLOCK

// HelperFunctions/F_ValidReqID
FUNCTION F_ValidReqID : BOOL
VAR_INPUT
    ReqID : DWORD;
END_VAR
VAR
END_VAR

F_ValidReqID := ReqID <> PMPS_GVL.EXCLUDED_ASSERTION_ID AND ReqID <> 0;

END_FUNCTION

// HelperFunctions/FB_DummyArbIO
(* Use to test other library integrations of PMPS preemptive functionality *)
(* This block stands in for the FB_SubSysToArb_IO block. *)

FUNCTION_BLOCK FB_DummyArbIO IMPLEMENTS I_HigherAuthority, I_LowerAuthority
VAR_INPUT
    //stCurrentBP : REFERENCE TO ST_BeamParams; //Set to something to redirect currentBP update
    LA : I_LowerAuthority;

    tRateDelay : TIME; // Delay until rate is looped back into q_stSimulatedBPReadback
    tTransDelay : TIME; // Delay until transmission is looped back into q_stSimulatedBPReadback
    tPEDelay : TIME; // Delay until PE is looped back into q_stSimulatedBPReadback
    tAptDelay : TIME; // Delay until apertures are looped back into q_stSimulatedBPReadback
    tSattDelay : TIME; // Delay until apertures are looped back into q_stSimulatedBPReadback

END_VAR
VAR_OUTPUT
    q_stSimulatedBPReadback : ST_BeamParams; // Updated to
END_VAR
VAR_IN_OUT
    FFO : FB_HardwareFFOutput;
END_VAR
VAR
   bAutoUpdateBP : BOOL := FALSE; // Set by AutoUpdateBP property, if true causes this FB to update PMPS_GVL.stCurrentBP to the
   // requested value automatically within the RequestBP method and restore it within the RemoveRequest method
   stNewReqBP : ST_BeamParams;

   stReqOutBP : ST_BeamParams;// To be written on next ApplyBPReq call

   stSaveCurrentBP : ST_BeamParams; // Will be restored after RemoveRequest then ApplyBPReq call

   nSavedID : DWORD; // Used to simulate CheckRequest method

   tonRate : TON;
   tonTrans : TON;
   tonPE : TON;
   tonApt : TON;
   tonSatt : TON;
   tonBCRange: TON;
   tonBC :TON;

END_VAR


LA.ElevateRequest(THIS^);

ApplyBPReq(FALSE); //If autoupdate is set, this will propagate the request to PMPS_GVL.stCurrentBP;

// Call this method to update q_stSimulatedBPReadback at will, used if auto-update is set to false
METHOD ApplyBPReq
VAR_INPUT
    bUpdateBP : BOOL := FALSE; // Set true and call this method to set q_stSimulatedBPReadback to the request
END_VAR
VAR
    BP : REFERENCE TO ST_BeamParams;
END_VAR

IF bUpdateBP THEN
    stSaveCurrentBP := q_stSimulatedBPReadback;
    q_stSimulatedBPReadback := stReqOutBP;
ELSIF bAutoUpdateBP THEN
    tonApt.IN := 0 <> MEMCMP(ADR(stReqOutBP.astApertures), ADR(q_stSimulatedBPReadback.astApertures), SIZEOF(q_stSimulatedBPReadback.astApertures));
    tonApt(PT:=tAptDelay);
    IF tonApt.Q THEN q_stSimulatedBPReadback.astApertures := stReqOutBP.astApertures; END_IF

    tonRate(IN:=stReqOutBP.nRate<>q_stSimulatedBPReadback.nRate, PT:=tRateDelay);
    IF tonRate.Q THEN q_stSimulatedBPReadback.nRate := stReqOutBP.nRate; END_IF

    tonTrans(IN:=stReqOutBP.nTran<>q_stSimulatedBPReadback.nTran, PT:=tTransDelay);
    IF tonTrans.Q THEN q_stSimulatedBPReadback.nTran := stReqOutBP.nTran; END_IF

    tonPE(IN:=stReqOutBP.neVRange<>q_stSimulatedBPReadback.neVRange, PT:=tPEDelay);
    IF tonPE.Q THEN
        IF stReqOutBP.neVRange = 0 THEN
            q_stSimulatedBPReadback.neVRange := 0;
            q_stSimulatedBPReadback.neVRange.0 := TRUE;
        ELSE
            q_stSimulatedBPReadback.neVRange := stReqOutBP.neVRange;
        END_IF
    END_IF

    tonBCRange(IN:=stReqOutBP.nBCRange<>q_stSimulatedBPReadback.nBCRange, PT:=tPEDelay);
     IF tonBCRange.Q THEN
        IF stReqOutBP.nBCRange = 0 THEN
            q_stSimulatedBPReadback.nBCRange := 0;
        ELSE
            q_stSimulatedBPReadback.nBCRange := stReqOutBP.nBCRange;
        END_IF
    END_IF

    tonSatt.IN := 0 <> MEMCMP(ADR(stReqOutBP.astAttenuators), ADR(q_stSimulatedBPReadback.astAttenuators), SIZEOF(q_stSimulatedBPReadback.astAttenuators));
    tonSatt(PT:=tSattDelay);
    IF tonSatt.Q THEN q_stSimulatedBPReadback.astAttenuators := stReqOutBP.astAttenuators; END_IF
END_IF

ffo.ExecuteNoLog();

IF NOT ffo.q_xFastFaultOut THEN q_stSimulatedBPReadback.nRate := 0; END_IF
END_METHOD

PROPERTY AutoUpdateBP : BOOL
GET
AutoUpdateBP := bAutoUpdateBP;
END_GET
SET
bAutoUpdateBP := AutoUpdateBP;
END_SET
END_PROPERTY

METHOD CheckRequest : BOOL
VAR_INPUT
    nReqID	: DWORD;
END_VAR
CheckRequest := nReqID = nSavedID AND (nReqID <> 0) AND (nReqID <> PMPS_GVL.EXCLUDED_ASSERTION_ID);
END_METHOD


METHOD RemoveRequest : BOOL
VAR_INPUT
    (*StateID to remove*)
    nReqID	: DWORD;
END_VAR

nSavedID := 0;

stReqOutBP := stSaveCurrentBP;

RemoveRequest := TRUE;
END_METHOD

// Request a BP from this higher authority
METHOD RequestBP : BOOL
VAR_INPUT
    (*StateID of state requesting beam parameter set*)
    nReqID	: DWORD;
    (*Requested beam params*)
    stReqBP	: ST_BeamParams;
END_VAR
IF nReqID <> 0 AND nReqID <> PMPS_GVL.EXCLUDED_ASSERTION_ID THEN
    nSavedID := nReqID;
    stReqOutBP := stReqBP;

    RequestBP := TRUE;
ELSE
    RequestBP := FALSE;
END_IF
END_METHOD

// <Arbiter Internal>
// Elevates the arbitrated BP set to something above.
// Could be another arbiter, or a BP requester/ IO,
// or an FB that locks in a specific portion of the BP set.
METHOD ElevateRequest : BOOL
VAR_INPUT
    HigherAuthority : I_HigherAuthority;
END_VAR
END_METHOD

PROPERTY nLowerAuthorityID : DWORD
GET
nLowerAuthorityID := PMPS_GVL.EXCLUDED_ASSERTION_ID;
END_GET
END_PROPERTY

END_FUNCTION_BLOCK

// MajorComponents/I_HigherAuthority
INTERFACE I_HigherAuthority

//Verify with this higher authority that the request is being included
METHOD CheckRequest : BOOL
VAR_INPUT
    nReqID    :    DWORD;
END_VAR
END_METHOD

//Remove the request from this higher authority
METHOD RemoveRequest : BOOL
VAR_INPUT
	nReqID    :    DWORD; //StateID to remove
END_VAR
END_METHOD

// Request a BP from this higher authority
METHOD RequestBP : BOOL
VAR_INPUT
    nReqID    :    DWORD; //StateID of state requesting beam parameter set
    stReqBP        :    ST_BeamParams; //Requested beam params
END_VAR
END_METHOD

END_INTERFACE

// MajorComponents/I_LowerAuthority
INTERFACE I_LowerAuthority

// <Arbiter Internal>
// Elevates the arbitrated BP set to something above.
// Could be another arbiter, or a BP requester/ IO, 
// or an FB that locks in a specific portion of the BP set.
METHOD ElevateRequest : BOOL 
VAR_INPUT
    HigherAuthority : I_HigherAuthority;
END_VAR
END_METHOD

PROPERTY nLowerAuthorityID : DWORD
GET
END_GET
END_PROPERTY

END_INTERFACE

// HelperFunctions/FB_DummyHA
FUNCTION_BLOCK FB_DummyHA IMPLEMENTS I_HigherAuthority, I_LowerAuthority
VAR_INPUT
    ReqAcknowledged : BOOL := TRUE; // Use to control when the HA CHeckRequest Returns TRUE
END_VAR
VAR_OUTPUT
END_VAR
VAR
END_VAR

METHOD CheckRequest : BOOL
VAR_INPUT
    nReqID	: DWORD;
END_VAR
CheckRequest := ReqAcknowledged;
END_METHOD

// <Arbiter Internal>
// Elevates the arbitrated BP set to something above.
// Could be another arbiter, or a BP requester/ IO,
// or an FB that locks in a specific portion of the BP set.
METHOD ElevateRequest : BOOL
VAR_INPUT
    HigherAuthority : I_HigherAuthority;
END_VAR
END_METHOD

PROPERTY nLowerAuthorityID : DWORD
GET
nLowerAuthorityID := PMPS_GVL.EXCLUDED_ASSERTION_ID;
END_GET
END_PROPERTY


METHOD RemoveRequest : BOOL
VAR_INPUT
    (*StateID to remove*)
    nReqID	: DWORD;
END_VAR
RemoveRequest := TRUE;
END_METHOD


METHOD RequestBP : BOOL
VAR_INPUT
    (*StateID of state requesting beam parameter set*)
    nReqID	: DWORD;
    (*Requested beam params*)
    stReqBP	: ST_BeamParams;
END_VAR
RequestBP := TRUE;
END_METHOD

END_FUNCTION_BLOCK

// HelperFunctions/PE_Ranges
// Does nothing other than set the gvl for photon energy bitmask to one of two constants, K or L.
// Workaround for compile defines not fully working for libraries at the time of writing this.
// Otherwise I would have just used the compile define in the GVL declaration.
FUNCTION_BLOCK PE_Ranges
VAR_INPUT
END_VAR
VAR_OUTPUT
END_VAR
VAR
END_VAR

METHOD FB_init : BOOL
VAR_INPUT
    bInitRetains : BOOL; // if TRUE, the retain variables are initialized (warm start / cold start)
    bInCopyCode : BOOL;  // if TRUE, the instance afterwards gets moved into the copy code (online change)
END_VAR
{IF defined (L)}
    PMPS_GVL.g_areVBoundaries := PMPS_GVL.g_areVBoundariesL;
{ELSIF defined (K)}
    PMPS_GVL.g_areVBoundaries := PMPS_GVL.g_areVBoundariesK;
{END_IF}
END_METHOD

END_FUNCTION_BLOCK

// ImplicitChecks/CheckBounds
// Implicitly generated code : DO NOT EDIT
FUNCTION CheckBounds : DINT
VAR_INPUT
    index, lower, upper: DINT;
END_VAR

// Implicitly generated code : Only an Implementation suggestion
{noflow}
IF  index < lower THEN
    CheckBounds := lower;
ELSIF  index > upper THEN
    CheckBounds := upper;
ELSE
    CheckBounds := index;
END_IF
{flow}

END_FUNCTION

// ImplicitChecks/CheckDivDInt
// Implicitly generated code : DO NOT EDIT
FUNCTION CheckDivDInt : DINT
VAR_INPUT
    divisor:DINT;
END_VAR

// Implicitly generated code : Only an Implementation suggestion
{noflow}
IF divisor = 0 THEN
    CheckDivDInt:=1;
ELSE
    CheckDivDInt:=divisor;
END_IF;
{flow}

END_FUNCTION

// ImplicitChecks/CheckDivLInt
// Implicitly generated code : DO NOT EDIT
FUNCTION CheckDivLInt : LINT
VAR_INPUT
    divisor:LINT;
END_VAR

// Implicitly generated code : Only an Implementation suggestion
{noflow}
IF divisor = 0 THEN
    CheckDivLInt:=1;
ELSE
    CheckDivLInt:=divisor;
END_IF;
{flow}

END_FUNCTION

// ImplicitChecks/CheckDivLReal
// Implicitly generated code : DO NOT EDIT
FUNCTION CheckDivLReal : LREAL
VAR_INPUT
    divisor:LREAL;
END_VAR

// Implicitly generated code : Only an Implementation suggestion
{noflow}
IF divisor = 0 THEN
    CheckDivLReal:=1;
ELSE
    CheckDivLReal:=divisor;
END_IF;
{flow}

END_FUNCTION

// ImplicitChecks/CheckDivReal
// Implicitly generated code : DO NOT EDIT
FUNCTION CheckDivReal : REAL
VAR_INPUT
    divisor:REAL;
END_VAR

// Implicitly generated code : Only an Implementation suggestion
{noflow}
IF divisor = 0 THEN
    CheckDivReal:=1;
ELSE
    CheckDivReal:=divisor;
END_IF;
{flow}

END_FUNCTION

// ImplicitChecks/CheckLRangeSigned
// Implicitly generated code : DO NOT EDIT
FUNCTION CheckLRangeSigned : LINT
VAR_INPUT
    value, lower, upper: LINT;
END_VAR

// Implicitly generated code : Only an Implementation suggestion
{noflow}
IF (value < lower) THEN
    CheckLRangeSigned := lower;
ELSIF(value > upper) THEN
    CheckLRangeSigned := upper;
ELSE
    CheckLRangeSigned := value;
END_IF

{flow}

END_FUNCTION

// ImplicitChecks/CheckLRangeUnsigned
// Implicitly generated code : DO NOT EDIT
FUNCTION CheckLRangeUnsigned : ULINT
VAR_INPUT
    value, lower, upper: ULINT;
END_VAR

// Implicitly generated code : Only an Implementation suggestion
{noflow}
IF (value < lower) THEN
    CheckLRangeUnsigned := lower;
ELSIF(value > upper) THEN
    CheckLRangeUnsigned := upper;
ELSE
    CheckLRangeUnsigned := value;
END_IF
{flow}

END_FUNCTION

// ImplicitChecks/CheckPointer
// Implicitly generated code : DO NOT EDIT
FUNCTION CheckPointer : POINTER TO BYTE
VAR_INPUT
    ptToTest : POINTER TO BYTE; // Destination address of the pointer
    iSize : DINT;		        // Size of the type the pointer points to. (e.g: 20 for POINTER TO ARRAY [0..9] OF INT)
    iGran : DINT;		        // Granularity of the pointer access. This is the size of the biggest non-structured data type in the type the pointer points to. (e.g: 2 for POINTER TO ARRAY [0..9] OF INT)
    bWrite: BOOL;		        // Indicates read or write Access. TRUE = write access.
END_VAR

// No standard way of implementation. Fill your own code here
CheckPointer := ptToTest;
{flow}

END_FUNCTION

// ImplicitChecks/CheckRangeSigned
// Implicitly generated code : DO NOT EDIT
FUNCTION CheckRangeSigned : DINT
VAR_INPUT
    value, lower, upper: DINT;
END_VAR

// Implicitly generated code : Only an Implementation suggestion
{noflow}
IF (value < lower) THEN
    CheckRangeSigned := lower;
ELSIF(value > upper) THEN
    CheckRangeSigned := upper;
ELSE
    CheckRangeSigned := value;
END_IF
{flow}

END_FUNCTION

// ImplicitChecks/CheckRangeUnsigned
// Implicitly generated code : DO NOT EDIT
FUNCTION CheckRangeUnsigned : UDINT
VAR_INPUT
    value, lower, upper: UDINT;
END_VAR

// Implicitly generated code : Only an Implementation suggestion
{noflow}
IF (value < lower) THEN
    CheckRangeUnsigned := lower;
ELSIF(value > upper) THEN
    CheckRangeUnsigned := upper;
ELSE
    CheckRangeUnsigned := value;
END_IF
{flow}

END_FUNCTION

// MajorComponents/Arbiter/FB_Arbiter
(* FB Arbiter
A. Wallace 2020-6-26

The arbiter primary objectives are:
- Provide a simple interface for devices to request beam parameter sets
- Provide a way for devices to verify their BPS is active in the arbiter
- Provide a way for devices remove their requests from evaluation
- Evaluate all active beam parameter requests registered with the aribiter,
to determine the safest combination of all sets, provide this set as an output.
- Do all of this with minimal overhead

To these ends, the arbiter uses a hash-table, the rows being a state-id as the key, and a corresponding
 beam parameter set to be evaluated against all the other sets (or rows), in the table.

